LIN {X 0,Y 301.791,Z 514.009,A -85,B 0,C 180,E1 15031.288,E2 15031.288} C_VEL
LIN {X 0,Y 301.177,Z 510.493,A -85,B 0,C 180,E1 15037.195,E2 15037.195} C_VEL
LIN {X 0,Y 300.944,Z 500.832,A -85,B 0,C 180,E1 15043.548,E2 15043.548} C_VEL
LIN {X 0,Y 302.786,Z 486.239,A -85,B 0,C 180,E1 15049.383,E2 15049.383} C_VEL
LIN {X 0,Y 307.108,Z 465.65,A -85,B 0,C 180,E1 15054.908,E2 15054.908} C_VEL
LIN {X 0,Y 312.998,Z 440.583,A -85,B 0,C 180,E1 15059.52,E2 15059.52} C_VEL
LIN {X 0,Y 319.157,Z 413.117,A -85,B 0,C 180,E1 15062.937,E2 15062.937} C_VEL
LIN {X 0,Y 324.854,Z 381.907,A -85,B 0,C 180,E1 15065.445,E2 15065.445} C_VEL
LIN {X 0,Y 326.72,Z 362.395,A -85,B 0,C 180,E1 15066.545,E2 15066.545} C_VEL
LIN {X 0,Y 316.647,Z 334.378,A -85,B 0,C 180,E1 15069.125,E2 15069.125} C_VEL
LIN {X 0,Y 302.51,Z 308.079,A -85,B 0,C 180,E1 15072.331,E2 15072.331} C_VEL
LIN {X 0,Y 294.858,Z 301.001,A -85,B 0,C 180,E1 15074.423,E2 15074.423} C_VEL
LIN {X 0,Y 289.746,Z 297.975,A -85,B 0,C 180,E1 15077.118,E2 15077.118} C_VEL
LIN {X 0,Y 289.332,Z 297.81,A -85,B 0,C 180,E1 15077.961,E2 15077.961} C_VEL
LIN {X 0,Y 289.637,Z 297.81,A -85,B 0,C 180,E1 15086.468,E2 15086.468} C_VEL
LIN {X 0,Y 289.839,Z 297.81,A -85,B 0,C 180,E1 15092.259,E2 15092.259} C_VEL
LIN {X 0,Y 290.263,Z 297.81,A -85,B 0,C 180,E1 15099.35,E2 15099.35} C_VEL
LIN {X 0,Y 290.729,Z 297.81,A -85,B 0,C 180,E1 15108.036,E2 15108.036} C_VEL
LIN {X 0,Y 291.615,Z 297.81,A -85,B 0,C 180,E1 15117.052,E2 15117.052} C_VEL
LIN {X 0,Y 291.518,Z 297.81,A -85,B 0,C 180,E1 15122.986,E2 15122.986} C_VEL
LIN {X 0,Y 290.857,Z 297.81,A -85,B 0,C 180,E1 15131.997,E2 15131.997} C_VEL
LIN {X 0,Y 290.685,Z 297.81,A -85,B 0,C 180,E1 15134.967,E2 15134.967} C_VEL
LIN {X 0,Y 293.021,Z 303.499,A -85,B 0,C 180,E1 15135.796,E2 15135.796} C_VEL
LIN {X 0,Y 305.082,Z 328.065,A -85,B 0,C 180,E1 15139.617,E2 15139.617} C_VEL
LIN {X 0,Y 311.989,Z 352.876,A -85,B 0,C 180,E1 15143.226,E2 15143.226} C_VEL
LIN {X 0,Y 313.291,Z 368.052,A -85,B 0,C 180,E1 15145.499,E2 15145.499} C_VEL
LIN {X 0,Y 307.869,Z 391.312,A -85,B 0,C 180,E1 15149.111,E2 15149.111} C_VEL
LIN {X 0,Y 302.987,Z 408.721,A -85,B 0,C 180,E1 15153.242,E2 15153.242} C_VEL
LIN {X 0,Y 298.665,Z 422.191,A -85,B 0,C 180,E1 15158.382,E2 15158.382} C_VEL
LIN {X 0,Y 296.439,Z 428.527,A -85,B 0,C 180,E1 15162.658,E2 15162.658} C_VEL
LIN {X 0,Y 294.718,Z 431.283,A -85,B 0,C 180,E1 15168.271,E2 15168.271} C_VEL
LIN {X 0,Y 294.669,Z 428.472,A -85,B 0,C 180,E1 15173.6,E2 15173.6} C_VEL
LIN {X 0,Y 296.07,Z 420.423,A -85,B 0,C 180,E1 15178.758,E2 15178.758} C_VEL
LIN {X 0,Y 298.582,Z 406.454,A -85,B 0,C 180,E1 15183.785,E2 15183.785} C_VEL
LIN {X 0,Y 302.074,Z 387.104,A -85,B 0,C 180,E1 15188.21,E2 15188.21} C_VEL
LIN {X 0,Y 305.829,Z 362.988,A -85,B 0,C 180,E1 15191.816,E2 15191.816} C_VEL
LIN {X 0,Y 306.003,Z 353.399,A -85,B 0,C 180,E1 15192.975,E2 15192.975} C_VEL
LIN {X 0,Y 303.879,Z 347.718,A -85,B 0,C 180,E1 15193.781,E2 15193.781} C_VEL
LIN {X 0,Y 302.697,Z 371.6,A -85,B 0,C 180,E1 15196.166,E2 15196.166} C_VEL
LIN {X 0,Y 300.079,Z 393.048,A -85,B 0,C 180,E1 15199.498,E2 15199.498} C_VEL
LIN {X 0,Y 297.619,Z 409.556,A -85,B 0,C 180,E1 15203.45,E2 15203.45} C_VEL
LIN {X 0,Y 295.778,Z 421.095,A -85,B 0,C 180,E1 15207.808,E2 15207.808} C_VEL
LIN {X 0,Y 294.658,Z 428.496,A -85,B 0,C 180,E1 15212.936,E2 15212.936} C_VEL
LIN {X 0,Y 294.506,Z 430.214,A -85,B 0,C 180,E1 15215.883,E2 15215.883} C_VEL
LIN {X 0,Y 294.768,Z 430.176,A -85,B 0,C 180,E1 15218.835,E2 15218.835} C_VEL
LIN {X 0,Y 296.42,Z 425.865,A -85,B 0,C 180,E1 15223.994,E2 15223.994} C_VEL
LIN {X 0,Y 299.258,Z 415.447,A -85,B 0,C 180,E1 15229.134,E2 15229.134} C_VEL
LIN {X 0,Y 302.774,Z 400.098,A -85,B 0,C 180,E1 15233.499,E2 15233.499} C_VEL
LIN {X 0,Y 306.689,Z 379.427,A -85,B 0,C 180,E1 15237.174,E2 15237.174} C_VEL
LIN {X 0,Y 309.289,Z 356.641,A -85,B 0,C 180,E1 15239.755,E2 15239.755} C_VEL
LIN {X 0,Y 303.855,Z 332.82,A -85,B 0,C 180,E1 15242.082,E2 15242.082} C_VEL
LIN {X 0,Y 289.715,Z 297.81,A -85,B 0,C 180,E1 15244.957,E2 15244.957} C_VEL
LIN {X 0,Y 289.4,Z 297.81,A -85,B 0,C 180,E1 15253.085,E2 15253.085} C_VEL
LIN {X 0,Y 289.499,Z 297.81,A -85,B 0,C 180,E1 15261.433,E2 15261.433} C_VEL
LIN {X 0,Y 289.619,Z 297.81,A -85,B 0,C 180,E1 15268.576,E2 15268.576} C_VEL
LIN {X 0,Y 290.019,Z 297.81,A -85,B 0,C 180,E1 15275.381,E2 15275.381} C_VEL
LIN {X 0,Y 290.399,Z 297.81,A -85,B 0,C 180,E1 15281.814,E2 15281.814} C_VEL
LIN {X 0,Y 290.916,Z 297.81,A -85,B 0,C 180,E1 15290.249,E2 15290.249} C_VEL
LIN {X 0,Y 291.631,Z 297.81,A -85,B 0,C 180,E1 15297.015,E2 15297.015} C_VEL
LIN {X 0,Y 291.57,Z 297.81,A -85,B 0,C 180,E1 15302.948,E2 15302.948} C_VEL
LIN {X 0,Y 290.904,Z 297.81,A -85,B 0,C 180,E1 15311.957,E2 15311.957} C_VEL
LIN {X 0,Y 290.36,Z 297.81,A -85,B 0,C 180,E1 15320.695,E2 15320.695} C_VEL
LIN {X 0,Y 289.868,Z 297.81,A -85,B 0,C 180,E1 15327.918,E2 15327.918} C_VEL
LIN {X 0,Y 289.6,Z 297.81,A -85,B 0,C 180,E1 15334.95,E2 15334.95} C_VEL
LIN {X 0,Y 289.442,Z 297.81,A -85,B 0,C 180,E1 15343.122,E2 15343.122} C_VEL
LIN {X 0,Y 289.776,Z 298.498,A -85,B 0,C 180,E1 15350.428,E2 15350.428} C_VEL
LIN {X 0,Y 309.953,Z 350.629,A -85,B 0,C 180,E1 15353.903,E2 15353.903} C_VEL
LIN {X 0,Y 313.87,Z 365.849,A -85,B 0,C 180,E1 15354.929,E2 15354.929} C_VEL
LIN {X 0,Y 309.878,Z 397.751,A -85,B 0,C 180,E1 15356.906,E2 15356.906} C_VEL
LIN {X 0,Y 304.908,Z 427.348,A -85,B 0,C 180,E1 15359.928,E2 15359.928} C_VEL
LIN {X 0,Y 300.107,Z 452.766,A -85,B 0,C 180,E1 15363.792,E2 15363.792} C_VEL
LIN {X 0,Y 295.894,Z 475.187,A -85,B 0,C 180,E1 15368.692,E2 15368.692} C_VEL
LIN {X 0,Y 293.627,Z 492.914,A -85,B 0,C 180,E1 15374.346,E2 15374.346} C_VEL
LIN {X 0,Y 293.234,Z 505.119,A -85,B 0,C 180,E1 15380.371,E2 15380.371} C_VEL
LIN {X 0,Y 293.771,Z 511.106,A -85,B 0,C 180,E1 15385.58,E2 15385.58} C_VEL
LIN {X 0,Y 294.167,Z 512.941,A -85,B 0,C 180,E1 15389.999,E2 15389.999} C_VEL
LIN {X 0,Y 293.543,Z 510.787,A -85,B 0,C 180,E1 15395.9,E2 15395.9} C_VEL
LIN {X 0,Y 292.981,Z 503.359,A -85,B 0,C 180,E1 15401.957,E2 15401.957} C_VEL
LIN {X 0,Y 294.232,Z 490.805,A -85,B 0,C 180,E1 15407.921,E2 15407.921} C_VEL
LIN {X 0,Y 298.019,Z 471.697,A -85,B 0,C 180,E1 15413.895,E2 15413.895} C_VEL
LIN {X 0,Y 304.002,Z 447.808,A -85,B 0,C 180,E1 15418.944,E2 15418.944} C_VEL
LIN {X 0,Y 310.758,Z 420.082,A -85,B 0,C 180,E1 15422.904,E2 15422.904} C_VEL
LIN {X 0,Y 316.915,Z 390.149,A -85,B 0,C 180,E1 15425.689,E2 15425.689} C_VEL
LIN {X 0,Y 320.12,Z 364.362,A -85,B 0,C 180,E1 15427.286,E2 15427.286} C_VEL
LIN {X 0,Y 310.556,Z 337.099,A -85,B 0,C 180,E1 15429.99,E2 15429.99} C_VEL
LIN {X 0,Y 295.545,Z 309.18,A -85,B 0,C 180,E1 15433.663,E2 15433.663} C_VEL
LIN {X 0,Y 289.738,Z 299.386,A -85,B 0,C 180,E1 15435.268,E2 15435.268} C_VEL
LIN {X 0,Y 289.539,Z 297.81,A -85,B 0,C 180,E1 15435.571,E2 15435.571} C_VEL
LIN {X 0,Y 289.332,Z 297.81,A -85,B 0,C 180,E1 15437.961,E2 15437.961} C_VEL
LIN {X 0,Y 286.749,Z 297.81,A -85,B 0,C 180,E1 15440.505,E2 15440.505} C_VEL
LIN {X 0,Y 281.458,Z 297.81,A -85,B 0,C 180,E1 15444.808,E2 15444.808} C_VEL
LIN {X 0,Y 281.799,Z 297.81,A -85,B 0,C 180,E1 15451.209,E2 15451.209} C_VEL
LIN {X 0,Y 282.166,Z 297.81,A -85,B 0,C 180,E1 15458.036,E2 15458.036} C_VEL
LIN {X 0,Y 282.566,Z 297.81,A -85,B 0,C 180,E1 15464.532,E2 15464.532} C_VEL
LIN {X 0,Y 283.042,Z 297.81,A -85,B 0,C 180,E1 15470.816,E2 15470.816} C_VEL
LIN {X 0,Y 283.684,Z 297.81,A -85,B 0,C 180,E1 15476.97,E2 15476.97} C_VEL
LIN {X 0,Y 283.594,Z 297.81,A -85,B 0,C 180,E1 15483.069,E2 15483.069} C_VEL
LIN {X 0,Y 283.112,Z 297.81,A -85,B 0,C 180,E1 15489.221,E2 15489.221} C_VEL
LIN {X 0,Y 282.852,Z 297.81,A -85,B 0,C 180,E1 15493.125,E2 15493.125} C_VEL
LIN {X 0,Y 285.066,Z 303.301,A -85,B 0,C 180,E1 15493.996,E2 15493.996} C_VEL
LIN {X 0,Y 296.674,Z 325.625,A -85,B 0,C 180,E1 15497.88,E2 15497.88} C_VEL
LIN {X 0,Y 304.058,Z 348.441,A -85,B 0,C 180,E1 15501.442,E2 15501.442} C_VEL
LIN {X 0,Y 306.68,Z 369.409,A -85,B 0,C 180,E1 15504.744,E2 15504.744} C_VEL
LIN {X 0,Y 300.833,Z 392.925,A -85,B 0,C 180,E1 15508.507,E2 15508.507} C_VEL
LIN {X 0,Y 295.699,Z 410.151,A -85,B 0,C 180,E1 15512.734,E2 15512.734} C_VEL
LIN {X 0,Y 291.189,Z 423.319,A -85,B 0,C 180,E1 15517.915,E2 15517.915} C_VEL
LIN {X 0,Y 288.516,Z 430.204,A -85,B 0,C 180,E1 15522.928,E2 15522.928} C_VEL
LIN {X 0,Y 287.048,Z 432.419,A -85,B 0,C 180,E1 15527.419,E2 15527.419} C_VEL
LIN {X 0,Y 286.705,Z 430.823,A -85,B 0,C 180,E1 15532.171,E2 15532.171} C_VEL
LIN {X 0,Y 287.863,Z 423.717,A -85,B 0,C 180,E1 15537.767,E2 15537.767} C_VEL
LIN {X 0,Y 290.131,Z 411.587,A -85,B 0,C 180,E1 15542.813,E2 15542.813} C_VEL
LIN {X 0,Y 293.356,Z 394.666,A -85,B 0,C 180,E1 15547.289,E2 15547.289} C_VEL
LIN {X 0,Y 297.189,Z 372.469,A -85,B 0,C 180,E1 15551.203,E2 15551.203} C_VEL
LIN {X 0,Y 298.833,Z 356.279,A -85,B 0,C 180,E1 15553.285,E2 15553.285} C_VEL
LIN {X 0,Y 296.944,Z 353.965,A -85,B 0,C 180,E1 15553.766,E2 15553.766} C_VEL
LIN {X 0,Y 294.567,Z 378.458,A -85,B 0,C 180,E1 15556.486,E2 15556.486} C_VEL
LIN {X 0,Y 291.698,Z 399.409,A -85,B 0,C 180,E1 15560.241,E2 15560.241} C_VEL
LIN {X 0,Y 289.176,Z 415.34,A -85,B 0,C 180,E1 15564.761,E2 15564.761} C_VEL
LIN {X 0,Y 287.366,Z 426.199,A -85,B 0,C 180,E1 15570.001,E2 15570.001} C_VEL
LIN {X 0,Y 286.828,Z 429.651,A -85,B 0,C 180,E1 15573.017,E2 15573.017} C_VEL
LIN {X 0,Y 286.689,Z 431.329,A -85,B 0,C 180,E1 15576.044,E2 15576.044} C_VEL
LIN {X 0,Y 287.015,Z 431.225,A -85,B 0,C 180,E1 15579.076,E2 15579.076} C_VEL
LIN {X 0,Y 288.731,Z 426.889,A -85,B 0,C 180,E1 15584.318,E2 15584.318} C_VEL
LIN {X 0,Y 291.271,Z 418.194,A -85,B 0,C 180,E1 15588.893,E2 15588.893} C_VEL
LIN {X 0,Y 295.038,Z 402.907,A -85,B 0,C 180,E1 15593.602,E2 15593.602} C_VEL
LIN {X 0,Y 299.062,Z 383.23,A -85,B 0,C 180,E1 15597.366,E2 15597.366} C_VEL
LIN {X 0,Y 302.392,Z 360.317,A -85,B 0,C 180,E1 15600.134,E2 15600.134} C_VEL
LIN {X 0,Y 297.677,Z 337.372,A -85,B 0,C 180,E1 15602.53,E2 15602.53} C_VEL
LIN {X 0,Y 285.512,Z 307.036,A -85,B 0,C 180,E1 15605.099,E2 15605.099} C_VEL
LIN {X 0,Y 281.647,Z 297.81,A -85,B 0,C 180,E1 15605.978,E2 15605.978} C_VEL
LIN {X 0,Y 281.379,Z 297.81,A -85,B 0,C 180,E1 15614.202,E2 15614.202} C_VEL
LIN {X 0,Y 281.401,Z 297.81,A -85,B 0,C 180,E1 15619.921,E2 15619.921} C_VEL
LIN {X 0,Y 281.677,Z 297.81,A -85,B 0,C 180,E1 15627.583,E2 15627.583} C_VEL
LIN {X 0,Y 282.132,Z 297.81,A -85,B 0,C 180,E1 15635.404,E2 15635.404} C_VEL
LIN {X 0,Y 282.555,Z 297.81,A -85,B 0,C 180,E1 15644.01,E2 15644.01} C_VEL
LIN {X 0,Y 283.082,Z 297.81,A -85,B 0,C 180,E1 15650.778,E2 15650.778} C_VEL
LIN {X 0,Y 283.701,Z 297.81,A -85,B 0,C 180,E1 15656.932,E2 15656.932} C_VEL
LIN {X 0,Y 283.645,Z 297.81,A -85,B 0,C 180,E1 15663.031,E2 15663.031} C_VEL
LIN {X 0,Y 283.152,Z 297.81,A -85,B 0,C 180,E1 15669.181,E2 15669.181} C_VEL
LIN {X 0,Y 282.614,Z 297.81,A -85,B 0,C 180,E1 15676.031,E2 15676.031} C_VEL
LIN {X 0,Y 282.143,Z 297.81,A -85,B 0,C 180,E1 15684.601,E2 15684.601} C_VEL
LIN {X 0,Y 281.742,Z 297.81,A -85,B 0,C 180,E1 15692.363,E2 15692.363} C_VEL
LIN {X 0,Y 281.432,Z 297.81,A -85,B 0,C 180,E1 15701.351,E2 15701.351} C_VEL
LIN {X 0,Y 281.777,Z 297.81,A -85,B 0,C 180,E1 15709.488,E2 15709.488} C_VEL
LIN {X 0,Y 302.846,Z 352.489,A -85,B 0,C 180,E1 15713.315,E2 15713.315} C_VEL
LIN {X 0,Y 306.58,Z 367.201,A -85,B 0,C 180,E1 15714.371,E2 15714.371} C_VEL
LIN {X 0,Y 302.451,Z 398.701,A -85,B 0,C 180,E1 15716.422,E2 15716.422} C_VEL
LIN {X 0,Y 297.175,Z 428.783,A -85,B 0,C 180,E1 15719.648,E2 15719.648} C_VEL
LIN {X 0,Y 291.863,Z 455.219,A -85,B 0,C 180,E1 15723.929,E2 15723.929} C_VEL
LIN {X 0,Y 287.627,Z 477.566,A -85,B 0,C 180,E1 15729.24,E2 15729.24} C_VEL
LIN {X 0,Y 285.642,Z 493.29,A -85,B 0,C 180,E1 15734.683,E2 15734.683} C_VEL
LIN {X 0,Y 285.406,Z 504.98,A -85,B 0,C 180,E1 15740.873,E2 15740.873} C_VEL
LIN {X 0,Y 285.932,Z 509.912,A -85,B 0,C 180,E1 15745.459,E2 15745.459} C_VEL
LIN {X 0,Y 286.352,Z 511.824,A -85,B 0,C 180,E1 15749.999,E2 15749.999} C_VEL
LIN {X 0,Y 286.049,Z 511.441,A -85,B 0,C 180,E1 15753.023,E2 15753.023} C_VEL
LIN {X 0,Y 285.263,Z 506.719,A -85,B 0,C 180,E1 15759.13,E2 15759.13} C_VEL
LIN {X 0,Y 285.53,Z 496.88,A -85,B 0,C 180,E1 15765.321,E2 15765.321} C_VEL
LIN {X 0,Y 288.492,Z 480.067,A -85,B 0,C 180,E1 15771.88,E2 15771.88} C_VEL
LIN {X 0,Y 293.941,Z 458.261,A -85,B 0,C 180,E1 15777.517,E2 15777.517} C_VEL
LIN {X 0,Y 300.68,Z 432.847,A -85,B 0,C 180,E1 15781.984,E2 15781.984} C_VEL
LIN {X 0,Y 307.715,Z 403.515,A -85,B 0,C 180,E1 15785.398,E2 15785.398} C_VEL
LIN {X 0,Y 313.552,Z 371.306,A -85,B 0,C 180,E1 15787.722,E2 15787.722} C_VEL
LIN {X 0,Y 313.18,Z 364.985,A -85,B 0,C 180,E1 15788.214,E2 15788.214} C_VEL
LIN {X 0,Y 304.443,Z 339.762,A -85,B 0,C 180,E1 15790.922,E2 15790.922} C_VEL
LIN {X 0,Y 290.715,Z 314.15,A -85,B 0,C 180,E1 15794.487,E2 15794.487} C_VEL
LIN {X 0,Y 283.669,Z 303.218,A -85,B 0,C 180,E1 15796.549,E2 15796.549} C_VEL
LIN {X 0,Y 281.52,Z 297.81,A -85,B 0,C 180,E1 15797.338,E2 15797.338} C_VEL
LIN {X 0,Y 281.458,Z 297.81,A -85,B 0,C 180,E1 15804.808,E2 15804.808} C_VEL
LIN {X 0,Y 279.049,Z 297.81,A -85,B 0,C 180,E1 15807.427,E2 15807.427} C_VEL
LIN {X 0,Y 273.871,Z 297.81,A -85,B 0,C 180,E1 15811.859,E2 15811.859} C_VEL
LIN {X 0,Y 274.257,Z 297.81,A -85,B 0,C 180,E1 15819.284,E2 15819.284} C_VEL
LIN {X 0,Y 274.794,Z 297.81,A -85,B 0,C 180,E1 15827.331,E2 15827.331} C_VEL
LIN {X 0,Y 275.365,Z 297.81,A -85,B 0,C 180,E1 15833.727,E2 15833.727} C_VEL
LIN {X 0,Y 275.921,Z 297.81,A -85,B 0,C 180,E1 15840.02,E2 15840.02} C_VEL
LIN {X 0,Y 275.224,Z 297.81,A -85,B 0,C 180,E1 15849.29,E2 15849.29} C_VEL
LIN {X 0,Y 275.008,Z 298.149,A -85,B 0,C 180,E1 15851.091,E2 15851.091} C_VEL
LIN {X 0,Y 277.4,Z 303.463,A -85,B 0,C 180,E1 15852.06,E2 15852.06} C_VEL
LIN {X 0,Y 288.452,Z 323.451,A -85,B 0,C 180,E1 15856.024,E2 15856.024} C_VEL
LIN {X 0,Y 296.621,Z 346.543,A -85,B 0,C 180,E1 15859.91,E2 15859.91} C_VEL
LIN {X 0,Y 300.124,Z 369.507,A -85,B 0,C 180,E1 15863.738,E2 15863.738} C_VEL
LIN {X 0,Y 294.43,Z 392.663,A -85,B 0,C 180,E1 15867.49,E2 15867.49} C_VEL
LIN {X 0,Y 289.022,Z 409.878,A -85,B 0,C 180,E1 15871.675,E2 15871.675} C_VEL
LIN {X 0,Y 284.51,Z 422.433,A -85,B 0,C 180,E1 15876.38,E2 15876.38} C_VEL
LIN {X 0,Y 281.403,Z 430.156,A -85,B 0,C 180,E1 15881.347,E2 15881.347} C_VEL
LIN {X 0,Y 279.75,Z 433.129,A -85,B 0,C 180,E1 15885.475,E2 15885.475} C_VEL
LIN {X 0,Y 278.854,Z 432.696,A -85,B 0,C 180,E1 15890.907,E2 15890.907} C_VEL
LIN {X 0,Y 279.687,Z 426.762,A -85,B 0,C 180,E1 15896.704,E2 15896.704} C_VEL
LIN {X 0,Y 281.935,Z 415.187,A -85,B 0,C 180,E1 15902.173,E2 15902.173} C_VEL
LIN {X 0,Y 285.175,Z 398.75,A -85,B 0,C 180,E1 15906.979,E2 15906.979} C_VEL
LIN {X 0,Y 289.128,Z 377.292,A -85,B 0,C 180,E1 15911.11,E2 15911.11} C_VEL
LIN {X 0,Y 291.378,Z 363.262,A -85,B 0,C 180,E1 15913.065,E2 15913.065} C_VEL
LIN {X 0,Y 289.197,Z 360.16,A -85,B 0,C 180,E1 15913.713,E2 15913.713} C_VEL
LIN {X 0,Y 286.517,Z 383.805,A -85,B 0,C 180,E1 15916.679,E2 15916.679} C_VEL
LIN {X 0,Y 283.656,Z 403.2,A -85,B 0,C 180,E1 15920.533,E2 15920.533} C_VEL
LIN {X 0,Y 281.397,Z 416.682,A -85,B 0,C 180,E1 15924.616,E2 15924.616} C_VEL
LIN {X 0,Y 279.532,Z 427.42,A -85,B 0,C 180,E1 15930.001,E2 15930.001} C_VEL
LIN {X 0,Y 278.989,Z 430.807,A -85,B 0,C 180,E1 15933.101,E2 15933.101} C_VEL
LIN {X 0,Y 278.866,Z 432.437,A -85,B 0,C 180,E1 15936.214,E2 15936.214} C_VEL
LIN {X 0,Y 279.242,Z 432.277,A -85,B 0,C 180,E1 15939.331,E2 15939.331} C_VEL
LIN {X 0,Y 281.209,Z 427.535,A -85,B 0,C 180,E1 15944.925,E2 15944.925} C_VEL
LIN {X 0,Y 284.336,Z 417.08,A -85,B 0,C 180,E1 15950.18,E2 15950.18} C_VEL
LIN {X 0,Y 288.308,Z 401.414,A -85,B 0,C 180,E1 15954.755,E2 15954.755} C_VEL
LIN {X 0,Y 292.539,Z 380.963,A -85,B 0,C 180,E1 15958.491,E2 15958.491} C_VEL
LIN {X 0,Y 295.194,Z 360.337,A -85,B 0,C 180,E1 15960.949,E2 15960.949} C_VEL
LIN {X 0,Y 289.798,Z 336.185,A -85,B 0,C 180,E1 15963.542,E2 15963.542} C_VEL
LIN {X 0,Y 277.11,Z 306.368,A -85,B 0,C 180,E1 15966.232,E2 15966.232} C_VEL
LIN {X 0,Y 273.604,Z 297.81,A -85,B 0,C 180,E1 15967.086,E2 15967.086} C_VEL
LIN {X 0,Y 273.468,Z 297.81,A -85,B 0,C 180,E1 15975.836,E2 15975.836} C_VEL
LIN {X 0,Y 273.461,Z 297.81,A -85,B 0,C 180,E1 15982.601,E2 15982.601} C_VEL
LIN {X 0,Y 273.808,Z 297.81,A -85,B 0,C 180,E1 15990.24,E2 15990.24} C_VEL
LIN {X 0,Y 274.292,Z 297.81,A -85,B 0,C 180,E1 15999.27,E2 15999.27} C_VEL
LIN {X 0,Y 274.844,Z 297.81,A -85,B 0,C 180,E1 16007.293,E2 16007.293} C_VEL
LIN {X 0,Y 275.393,Z 297.81,A -85,B 0,C 180,E1 16013.688,E2 16013.688} C_VEL
LIN {X 0,Y 276.036,Z 297.81,A -85,B 0,C 180,E1 16019.98,E2 16019.98} C_VEL
LIN {X 0,Y 275.2,Z 297.81,A -85,B 0,C 180,E1 16029.449,E2 16029.449} C_VEL
LIN {X 0,Y 274.728,Z 297.81,A -85,B 0,C 180,E1 16035.92,E2 16035.92} C_VEL
LIN {X 0,Y 274.265,Z 297.81,A -85,B 0,C 180,E1 16042.632,E2 16042.632} C_VEL
LIN {X 0,Y 273.874,Z 297.81,A -85,B 0,C 180,E1 16049.706,E2 16049.706} C_VEL
LIN {X 0,Y 273.506,Z 297.81,A -85,B 0,C 180,E1 16057.342,E2 16057.342} C_VEL
LIN {X 0,Y 273.573,Z 297.81,A -85,B 0,C 180,E1 16065.786,E2 16065.786} C_VEL
LIN {X 0,Y 273.819,Z 297.81,A -85,B 0,C 180,E1 16068.497,E2 16068.497} C_VEL
LIN {X 0,Y 295.092,Z 352.338,A -85,B 0,C 180,E1 16072.563,E2 16072.563} C_VEL
LIN {X 0,Y 299.245,Z 369.351,A -85,B 0,C 180,E1 16073.843,E2 16073.843} C_VEL
LIN {X 0,Y 294.934,Z 400.043,A -85,B 0,C 180,E1 16075.971,E2 16075.971} C_VEL
LIN {X 0,Y 289.575,Z 429.128,A -85,B 0,C 180,E1 16079.223,E2 16079.223} C_VEL
LIN {X 0,Y 284.164,Z 455.141,A -85,B 0,C 180,E1 16083.593,E2 16083.593} C_VEL
LIN {X 0,Y 279.809,Z 477.301,A -85,B 0,C 180,E1 16089.066,E2 16089.066} C_VEL
LIN {X 0,Y 277.691,Z 493.638,A -85,B 0,C 180,E1 16095.041,E2 16095.041} C_VEL
LIN {X 0,Y 277.595,Z 504.699,A -85,B 0,C 180,E1 16101.402,E2 16101.402} C_VEL
LIN {X 0,Y 278.299,Z 509.701,A -85,B 0,C 180,E1 16106.891,E2 16106.891} C_VEL
LIN {X 0,Y 278.524,Z 510.7,A -85,B 0,C 180,E1 16109.999,E2 16109.999} C_VEL
LIN {X 0,Y 278.197,Z 510.343,A -85,B 0,C 180,E1 16113.108,E2 16113.108} C_VEL
LIN {X 0,Y 277.346,Z 505.67,A -85,B 0,C 180,E1 16119.393,E2 16119.393} C_VEL
LIN {X 0,Y 277.724,Z 495.895,A -85,B 0,C 180,E1 16125.763,E2 16125.763} C_VEL
LIN {X 0,Y 280.964,Z 479.199,A -85,B 0,C 180,E1 16132.485,E2 16132.485} C_VEL
LIN {X 0,Y 286.783,Z 457.502,A -85,B 0,C 180,E1 16138.265,E2 16138.265} C_VEL
LIN {X 0,Y 293.959,Z 432.034,A -85,B 0,C 180,E1 16142.833,E2 16142.833} C_VEL
LIN {X 0,Y 301.26,Z 403.104,A -85,B 0,C 180,E1 16146.275,E2 16146.275} C_VEL
LIN {X 0,Y 307.338,Z 371.242,A -85,B 0,C 180,E1 16148.624,E2 16148.624} C_VEL
LIN {X 0,Y 301.194,Z 349.042,A -85,B 0,C 180,E1 16151.067,E2 16151.067} C_VEL
LIN {X 0,Y 288.211,Z 322.64,A -85,B 0,C 180,E1 16154.706,E2 16154.706} C_VEL
LIN {X 0,Y 276.575,Z 304.046,A -85,B 0,C 180,E1 16158.362,E2 16158.362} C_VEL
LIN {X 0,Y 273.66,Z 299.357,A -85,B 0,C 180,E1 16159.406,E2 16159.406} C_VEL
LIN {X 0,Y 273.505,Z 297.81,A -85,B 0,C 180,E1 16159.647,E2 16159.647} C_VEL
LIN {X 0,Y 273.635,Z 297.81,A -85,B 0,C 180,E1 16166.555,E2 16166.555} C_VEL
LIN {X 0,Y 273.871,Z 297.81,A -85,B 0,C 180,E1 16171.859,E2 16171.859} C_VEL
LIN {X 0,Y 271.322,Z 297.81,A -85,B 0,C 180,E1 16174.572,E2 16174.572} C_VEL
LIN {X 0,Y 266.238,Z 297.81,A -85,B 0,C 180,E1 16179.168,E2 16179.168} C_VEL
LIN {X 0,Y 266.821,Z 297.81,A -85,B 0,C 180,E1 16186.946,E2 16186.946} C_VEL
LIN {X 0,Y 267.424,Z 297.81,A -85,B 0,C 180,E1 16193.54,E2 16193.54} C_VEL
LIN {X 0,Y 268.014,Z 297.81,A -85,B 0,C 180,E1 16200.02,E2 16200.02} C_VEL
LIN {X 0,Y 267.307,Z 297.81,A -85,B 0,C 180,E1 16208.683,E2 16208.683} C_VEL
LIN {X 0,Y 269.585,Z 303.422,A -85,B 0,C 180,E1 16209.789,E2 16209.789} C_VEL
LIN {X 0,Y 278.977,Z 319.201,A -85,B 0,C 180,E1 16213.472,E2 16213.472} C_VEL
LIN {X 0,Y 288.438,Z 342.011,A -85,B 0,C 180,E1 16217.789,E2 16217.789} C_VEL
LIN {X 0,Y 292.923,Z 364.093,A -85,B 0,C 180,E1 16221.632,E2 16221.632} C_VEL
LIN {X 0,Y 292.974,Z 375.24,A -85,B 0,C 180,E1 16223.547,E2 16223.547} C_VEL
LIN {X 0,Y 286.411,Z 397.791,A -85,B 0,C 180,E1 16227.545,E2 16227.545} C_VEL
LIN {X 0,Y 280.635,Z 414.67,A -85,B 0,C 180,E1 16232.171,E2 16232.171} C_VEL
LIN {X 0,Y 275.808,Z 426.847,A -85,B 0,C 180,E1 16237.603,E2 16237.603} C_VEL
LIN {X 0,Y 273.52,Z 431.879,A -85,B 0,C 180,E1 16241.483,E2 16241.483} C_VEL
LIN {X 0,Y 271.696,Z 434.557,A -85,B 0,C 180,E1 16246.252,E2 16246.252} C_VEL
LIN {X 0,Y 271.151,Z 432.168,A -85,B 0,C 180,E1 16253.146,E2 16253.146} C_VEL
LIN {X 0,Y 272.729,Z 423.507,A -85,B 0,C 180,E1 16259.28,E2 16259.28} C_VEL
LIN {X 0,Y 275.404,Z 410.394,A -85,B 0,C 180,E1 16264.442,E2 16264.442} C_VEL
LIN {X 0,Y 279.298,Z 391.265,A -85,B 0,C 180,E1 16269.259,E2 16269.259} C_VEL
LIN {X 0,Y 283.411,Z 368.522,A -85,B 0,C 180,E1 16273.058,E2 16273.058} C_VEL
LIN {X 0,Y 281.302,Z 366.516,A -85,B 0,C 180,E1 16273.728,E2 16273.728} C_VEL
LIN {X 0,Y 278.314,Z 389.906,A -85,B 0,C 180,E1 16277.077,E2 16277.077} C_VEL
LIN {X 0,Y 275.332,Z 408.596,A -85,B 0,C 180,E1 16281.332,E2 16281.332} C_VEL
LIN {X 0,Y 272.913,Z 421.74,A -85,B 0,C 180,E1 16286.038,E2 16286.038} C_VEL
LIN {X 0,Y 271.396,Z 430.54,A -85,B 0,C 180,E1 16291.594,E2 16291.594} C_VEL
LIN {X 0,Y 271.049,Z 433.537,A -85,B 0,C 180,E1 16296.394,E2 16296.394} C_VEL
LIN {X 0,Y 271.491,Z 433.327,A -85,B 0,C 180,E1 16299.6,E2 16299.6} C_VEL
LIN {X 0,Y 273.362,Z 429.156,A -85,B 0,C 180,E1 16304.852,E2 16304.852} C_VEL
LIN {X 0,Y 276.33,Z 419.884,A -85,B 0,C 180,E1 16309.957,E2 16309.957} C_VEL
LIN {X 0,Y 280.444,Z 404.981,A -85,B 0,C 180,E1 16314.718,E2 16314.718} C_VEL
LIN {X 0,Y 284.633,Z 386.282,A -85,B 0,C 180,E1 16318.5,E2 16318.5} C_VEL
LIN {X 0,Y 288.298,Z 363.539,A -85,B 0,C 180,E1 16321.425,E2 16321.425} C_VEL
LIN {X 0,Y 283.612,Z 340.371,A -85,B 0,C 180,E1 16324.067,E2 16324.067} C_VEL
LIN {X 0,Y 272.3,Z 312.387,A -85,B 0,C 180,E1 16326.721,E2 16326.721} C_VEL
LIN {X 0,Y 265.592,Z 297.81,A -85,B 0,C 180,E1 16328.305,E2 16328.305} C_VEL
LIN {X 0,Y 265.529,Z 297.81,A -85,B 0,C 180,E1 16336.974,E2 16336.974} C_VEL
LIN {X 0,Y 265.597,Z 297.81,A -85,B 0,C 180,E1 16345.353,E2 16345.353} C_VEL
LIN {X 0,Y 265.986,Z 297.81,A -85,B 0,C 180,E1 16352.985,E2 16352.985} C_VEL
LIN {X 0,Y 266.451,Z 297.81,A -85,B 0,C 180,E1 16360.113,E2 16360.113} C_VEL
LIN {X 0,Y 266.873,Z 297.81,A -85,B 0,C 180,E1 16366.907,E2 16366.907} C_VEL
LIN {X 0,Y 267.453,Z 297.81,A -85,B 0,C 180,E1 16373.5,E2 16373.5} C_VEL
LIN {X 0,Y 268.128,Z 297.81,A -85,B 0,C 180,E1 16379.98,E2 16379.98} C_VEL
LIN {X 0,Y 267.481,Z 297.81,A -85,B 0,C 180,E1 16386.458,E2 16386.458} C_VEL
LIN {X 0,Y 266.991,Z 297.81,A -85,B 0,C 180,E1 16393.046,E2 16393.046} C_VEL
LIN {X 0,Y 266.492,Z 297.81,A -85,B 0,C 180,E1 16399.841,E2 16399.841} C_VEL
LIN {X 0,Y 266.011,Z 297.81,A -85,B 0,C 180,E1 16406.967,E2 16406.967} C_VEL
LIN {X 0,Y 265.66,Z 297.81,A -85,B 0,C 180,E1 16414.589,E2 16414.589} C_VEL
LIN {X 0,Y 265.587,Z 297.81,A -85,B 0,C 180,E1 16422.959,E2 16422.959} C_VEL
LIN {X 0,Y 265.766,Z 297.916,A -85,B 0,C 180,E1 16427.544,E2 16427.544} C_VEL
LIN {X 0,Y 287.407,Z 352.313,A -85,B 0,C 180,E1 16431.778,E2 16431.778} C_VEL
LIN {X 0,Y 292.004,Z 370.477,A -85,B 0,C 180,E1 16433.24,E2 16433.24} C_VEL
LIN {X 0,Y 287.229,Z 402.531,A -85,B 0,C 180,E1 16435.613,E2 16435.613} C_VEL
LIN {X 0,Y 281.418,Z 431.954,A -85,B 0,C 180,E1 16439.155,E2 16439.155} C_VEL
LIN {X 0,Y 276.038,Z 456.758,A -85,B 0,C 180,E1 16443.629,E2 16443.629} C_VEL
LIN {X 0,Y 271.74,Z 478.163,A -85,B 0,C 180,E1 16449.266,E2 16449.266} C_VEL
LIN {X 0,Y 269.756,Z 493.932,A -85,B 0,C 180,E1 16455.419,E2 16455.419} C_VEL
LIN {X 0,Y 269.828,Z 504.415,A -85,B 0,C 180,E1 16461.962,E2 16461.962} C_VEL
LIN {X 0,Y 270.455,Z 508.519,A -85,B 0,C 180,E1 16466.801,E2 16466.801} C_VEL
LIN {X 0,Y 270.722,Z 509.579,A -85,B 0,C 180,E1 16469.999,E2 16469.999} C_VEL
LIN {X 0,Y 270.332,Z 509.234,A -85,B 0,C 180,E1 16473.199,E2 16473.199} C_VEL
LIN {X 0,Y 269.466,Z 504.635,A -85,B 0,C 180,E1 16479.671,E2 16479.671} C_VEL
LIN {X 0,Y 270.117,Z 493.686,A -85,B 0,C 180,E1 16486.858,E2 16486.858} C_VEL
LIN {X 0,Y 273.711,Z 477.349,A -85,B 0,C 180,E1 16493.464,E2 16493.464} C_VEL
LIN {X 0,Y 279.697,Z 456.738,A -85,B 0,C 180,E1 16499.048,E2 16499.048} C_VEL
LIN {X 0,Y 287.234,Z 431.473,A -85,B 0,C 180,E1 16503.703,E2 16503.703} C_VEL
LIN {X 0,Y 294.896,Z 402.74,A -85,B 0,C 180,E1 16507.188,E2 16507.188} C_VEL
LIN {X 0,Y 300.892,Z 371.688,A -85,B 0,C 180,E1 16509.577,E2 16509.577} C_VEL
LIN {X 0,Y 293.59,Z 347.701,A -85,B 0,C 180,E1 16512.527,E2 16512.527} C_VEL
LIN {X 0,Y 280.155,Z 321.431,A -85,B 0,C 180,E1 16516.651,E2 16516.651} C_VEL
LIN {X 0,Y 268.475,Z 303.948,A -85,B 0,C 180,E1 16520.776,E2 16520.776} C_VEL
LIN {X 0,Y 265.627,Z 298.934,A -85,B 0,C 180,E1 16521.996,E2 16521.996} C_VEL
LIN {X 0,Y 265.574,Z 297.81,A -85,B 0,C 180,E1 16522.446,E2 16522.446} C_VEL
LIN {X 0,Y 265.775,Z 297.81,A -85,B 0,C 180,E1 16529.292,E2 16529.292} C_VEL
LIN {X 0,Y 266.179,Z 297.81,A -85,B 0,C 180,E1 16536.641,E2 16536.641} C_VEL
LIN {X 0,Y 266.238,Z 297.81,A -85,B 0,C 180,E1 16539.168,E2 16539.168} C_VEL
LIN {X 0,Y 264.072,Z 297.81,A -85,B 0,C 180,E1 16541.953,E2 16541.953} C_VEL
LIN {X 0,Y 258.879,Z 297.81,A -85,B 0,C 180,E1 16546.674,E2 16546.674} C_VEL
LIN {X 0,Y 259.474,Z 297.81,A -85,B 0,C 180,E1 16553.341,E2 16553.341} C_VEL
LIN {X 0,Y 260.106,Z 297.81,A -85,B 0,C 180,E1 16560.021,E2 16560.021} C_VEL
LIN {X 0,Y 259.571,Z 297.883,A -85,B 0,C 180,E1 16565.86,E2 16565.86} C_VEL
LIN {X 0,Y 261.491,Z 303.044,A -85,B 0,C 180,E1 16566.992,E2 16566.992} C_VEL
LIN {X 0,Y 264.165,Z 306.401,A -85,B 0,C 180,E1 16568.206,E2 16568.206} C_VEL
LIN {X 0,Y 275.569,Z 326.661,A -85,B 0,C 180,E1 16573.205,E2 16573.205} C_VEL
LIN {X 0,Y 283.292,Z 348.205,A -85,B 0,C 180,E1 16577.454,E2 16577.454} C_VEL
LIN {X 0,Y 286.745,Z 370.855,A -85,B 0,C 180,E1 16581.636,E2 16581.636} C_VEL
LIN {X 0,Y 285.636,Z 379.889,A -85,B 0,C 180,E1 16583.169,E2 16583.169} C_VEL
LIN {X 0,Y 278.979,Z 401.075,A -85,B 0,C 180,E1 16587.211,E2 16587.211} C_VEL
LIN {X 0,Y 272.678,Z 417.898,A -85,B 0,C 180,E1 16592.237,E2 16592.237} C_VEL
LIN {X 0,Y 267.782,Z 429.298,A -85,B 0,C 180,E1 16597.917,E2 16597.917} C_VEL
LIN {X 0,Y 264.948,Z 434.582,A -85,B 0,C 180,E1 16603.144,E2 16603.144} C_VEL
LIN {X 0,Y 263.487,Z 435.76,A -85,B 0,C 180,E1 16608.15,E2 16608.15} C_VEL
LIN {X 0,Y 263.343,Z 433.024,A -85,B 0,C 180,E1 16613.38,E2 16613.38} C_VEL
LIN {X 0,Y 264.827,Z 425.093,A -85,B 0,C 180,E1 16619.149,E2 16619.149} C_VEL
LIN {X 0,Y 267.562,Z 412.143,A -85,B 0,C 180,E1 16624.522,E2 16624.522} C_VEL
LIN {X 0,Y 271.56,Z 393.392,A -85,B 0,C 180,E1 16629.479,E2 16629.479} C_VEL
LIN {X 0,Y 274.804,Z 372.608,A -85,B 0,C 180,E1 16633.246,E2 16633.246} C_VEL
LIN {X 0,Y 273.498,Z 371.778,A -85,B 0,C 180,E1 16633.679,E2 16633.679} C_VEL
LIN {X 0,Y 270.462,Z 393.508,A -85,B 0,C 180,E1 16637.105,E2 16637.105} C_VEL
LIN {X 0,Y 267.323,Z 411.839,A -85,B 0,C 180,E1 16641.643,E2 16641.643} C_VEL
LIN {X 0,Y 264.808,Z 424.675,A -85,B 0,C 180,E1 16646.734,E2 16646.734} C_VEL
LIN {X 0,Y 263.575,Z 431.714,A -85,B 0,C 180,E1 16651.641,E2 16651.641} C_VEL
LIN {X 0,Y 263.232,Z 434.632,A -85,B 0,C 180,E1 16656.584,E2 16656.584} C_VEL
LIN {X 0,Y 264.216,Z 433.6,A -85,B 0,C 180,E1 16661.532,E2 16661.532} C_VEL
LIN {X 0,Y 266.792,Z 427.234,A -85,B 0,C 180,E1 16667.275,E2 16667.275} C_VEL
LIN {X 0,Y 270.504,Z 415.399,A -85,B 0,C 180,E1 16672.553,E2 16672.553} C_VEL
LIN {X 0,Y 274.911,Z 399.231,A -85,B 0,C 180,E1 16676.927,E2 16676.927} C_VEL
LIN {X 0,Y 279.383,Z 378.287,A -85,B 0,C 180,E1 16680.537,E2 16680.537} C_VEL
LIN {X 0,Y 281.038,Z 362.366,A -85,B 0,C 180,E1 16682.476,E2 16682.476} C_VEL
LIN {X 0,Y 275.582,Z 338.585,A -85,B 0,C 180,E1 16685.256,E2 16685.256} C_VEL
LIN {X 0,Y 262.275,Z 308.128,A -85,B 0,C 180,E1 16688.36,E2 16688.36} C_VEL
LIN {X 0,Y 257.58,Z 297.81,A -85,B 0,C 180,E1 16689.671,E2 16689.671} C_VEL
LIN {X 0,Y 257.476,Z 297.81,A -85,B 0,C 180,E1 16695.277,E2 16695.277} C_VEL
LIN {X 0,Y 257.615,Z 297.81,A -85,B 0,C 180,E1 16704.116,E2 16704.116} C_VEL
LIN {X 0,Y 257.917,Z 297.81,A -85,B 0,C 180,E1 16712.067,E2 16712.067} C_VEL
LIN {X 0,Y 258.429,Z 297.81,A -85,B 0,C 180,E1 16719.469,E2 16719.469} C_VEL
LIN {X 0,Y 258.938,Z 297.81,A -85,B 0,C 180,E1 16726.498,E2 16726.498} C_VEL
LIN {X 0,Y 259.502,Z 297.81,A -85,B 0,C 180,E1 16733.432,E2 16733.432} C_VEL
LIN {X 0,Y 260.219,Z 297.81,A -85,B 0,C 180,E1 16739.979,E2 16739.979} C_VEL
LIN {X 0,Y 259.346,Z 297.81,A -85,B 0,C 180,E1 16748.446,E2 16748.446} C_VEL
LIN {X 0,Y 258.742,Z 297.81,A -85,B 0,C 180,E1 16756.933,E2 16756.933} C_VEL
LIN {X 0,Y 258.243,Z 297.81,A -85,B 0,C 180,E1 16764.122,E2 16764.122} C_VEL
LIN {X 0,Y 257.808,Z 297.81,A -85,B 0,C 180,E1 16771.765,E2 16771.765} C_VEL
LIN {X 0,Y 257.537,Z 297.81,A -85,B 0,C 180,E1 16780.383,E2 16780.383} C_VEL
LIN {X 0,Y 257.714,Z 297.81,A -85,B 0,C 180,E1 16786.467,E2 16786.467} C_VEL
LIN {X 0,Y 278.795,Z 349.569,A -85,B 0,C 180,E1 16790.747,E2 16790.747} C_VEL
LIN {X 0,Y 284.759,Z 371.949,A -85,B 0,C 180,E1 16792.631,E2 16792.631} C_VEL
LIN {X 0,Y 279.844,Z 403.041,A -85,B 0,C 180,E1 16795.044,E2 16795.044} C_VEL
LIN {X 0,Y 273.806,Z 432.344,A -85,B 0,C 180,E1 16798.719,E2 16798.719} C_VEL
LIN {X 0,Y 267.956,Z 458.32,A -85,B 0,C 180,E1 16803.664,E2 16803.664} C_VEL
LIN {X 0,Y 263.657,Z 478.957,A -85,B 0,C 180,E1 16809.478,E2 16809.478} C_VEL
LIN {X 0,Y 261.816,Z 494.089,A -85,B 0,C 180,E1 16815.82,E2 16815.82} C_VEL
LIN {X 0,Y 261.955,Z 503.128,A -85,B 0,C 180,E1 16821.719,E2 16821.719} C_VEL
LIN {X 0,Y 262.609,Z 507.333,A -85,B 0,C 180,E1 16826.705,E2 16826.705} C_VEL
LIN {X 0,Y 262.891,Z 508.452,A -85,B 0,C 180,E1 16829.999,E2 16829.999} C_VEL
LIN {X 0,Y 262.474,Z 508.125,A -85,B 0,C 180,E1 16833.295,E2 16833.295} C_VEL
LIN {X 0,Y 261.556,Z 503.605,A -85,B 0,C 180,E1 16839.966,E2 16839.966} C_VEL
LIN {X 0,Y 262.351,Z 492.862,A -85,B 0,C 180,E1 16847.312,E2 16847.312} C_VEL
LIN {X 0,Y 266.121,Z 477.071,A -85,B 0,C 180,E1 16853.969,E2 16853.969} C_VEL
LIN {X 0,Y 272.682,Z 456.043,A -85,B 0,C 180,E1 16859.87,E2 16859.87} C_VEL
LIN {X 0,Y 280.623,Z 430.934,A -85,B 0,C 180,E1 16864.608,E2 16864.608} C_VEL
LIN {X 0,Y 288.768,Z 401.849,A -85,B 0,C 180,E1 16868.206,E2 16868.206} C_VEL
LIN {X 0,Y 294.466,Z 373.099,A -85,B 0,C 180,E1 16870.52,E2 16870.52} C_VEL
LIN {X 0,Y 287.061,Z 348.85,A -85,B 0,C 180,E1 16873.775,E2 16873.775} C_VEL
LIN {X 0,Y 273.819,Z 323.115,A -85,B 0,C 180,E1 16878.246,E2 16878.246} C_VEL
LIN {X 0,Y 264.129,Z 309.19,A -85,B 0,C 180,E1 16881.944,E2 16881.944} C_VEL
LIN {X 0,Y 260.929,Z 304.218,A -85,B 0,C 180,E1 16883.4,E2 16883.4} C_VEL
LIN {X 0,Y 257.842,Z 299.269,A -85,B 0,C 180,E1 16884.952,E2 16884.952} C_VEL
LIN {X 0,Y 257.729,Z 297.81,A -85,B 0,C 180,E1 16885.333,E2 16885.333} C_VEL
LIN {X 0,Y 257.923,Z 297.81,A -85,B 0,C 180,E1 16892.115,E2 16892.115} C_VEL
LIN {X 0,Y 258.383,Z 297.81,A -85,B 0,C 180,E1 16899.509,E2 16899.509} C_VEL
LIN {X 0,Y 258.879,Z 297.81,A -85,B 0,C 180,E1 16906.674,E2 16906.674} C_VEL
LIN {X 0,Y 256.455,Z 297.81,A -85,B 0,C 180,E1 16909.533,E2 16909.533} C_VEL
LIN {X 0,Y 251.582,Z 297.81,A -85,B 0,C 180,E1 16914.383,E2 16914.383} C_VEL
LIN {X 0,Y 251.965,Z 297.81,A -85,B 0,C 180,E1 16921.737,E2 16921.737} C_VEL
LIN {X 0,Y 251.955,Z 298.668,A -85,B 0,C 180,E1 16922.489,E2 16922.489} C_VEL
LIN {X 0,Y 254.902,Z 304.087,A -85,B 0,C 180,E1 16924.371,E2 16924.371} C_VEL
LIN {X 0,Y 256.727,Z 306.559,A -85,B 0,C 180,E1 16925.376,E2 16925.376} C_VEL
LIN {X 0,Y 265.264,Z 320.726,A -85,B 0,C 180,E1 16929.642,E2 16929.642} C_VEL
LIN {X 0,Y 273.598,Z 338.927,A -85,B 0,C 180,E1 16933.984,E2 16933.984} C_VEL
LIN {X 0,Y 279.101,Z 360.562,A -85,B 0,C 180,E1 16938.337,E2 16938.337} C_VEL
LIN {X 0,Y 280.254,Z 377.954,A -85,B 0,C 180,E1 16941.748,E2 16941.748} C_VEL
LIN {X 0,Y 272.753,Z 400.941,A -85,B 0,C 180,E1 16946.056,E2 16946.056} C_VEL
LIN {X 0,Y 266.082,Z 417.996,A -85,B 0,C 180,E1 16951.093,E2 16951.093} C_VEL
LIN {X 0,Y 261.291,Z 428.477,A -85,B 0,C 180,E1 16956.05,E2 16956.05} C_VEL
LIN {X 0,Y 258.357,Z 434.177,A -85,B 0,C 180,E1 16960.599,E2 16960.599} C_VEL
LIN {X 0,Y 256.412,Z 436.733,A -85,B 0,C 180,E1 16965.074,E2 16965.074} C_VEL
LIN {X 0,Y 255.391,Z 435.167,A -85,B 0,C 180,E1 16972.042,E2 16972.042} C_VEL
LIN {X 0,Y 256.542,Z 428.336,A -85,B 0,C 180,E1 16978.037,E2 16978.037} C_VEL
LIN {X 0,Y 259.143,Z 416.569,A -85,B 0,C 180,E1 16983.632,E2 16983.632} C_VEL
LIN {X 0,Y 263.124,Z 398.605,A -85,B 0,C 180,E1 16988.98,E2 16988.98} C_VEL
LIN {X 0,Y 267.024,Z 377.568,A -85,B 0,C 180,E1 16993.166,E2 16993.166} C_VEL
LIN {X 0,Y 265.648,Z 376.608,A -85,B 0,C 180,E1 16993.607,E2 16993.607} C_VEL
LIN {X 0,Y 262.58,Z 397.042,A -85,B 0,C 180,E1 16997.134,E2 16997.134} C_VEL
LIN {X 0,Y 259.269,Z 414.876,A -85,B 0,C 180,E1 17001.929,E2 17001.929} C_VEL
LIN {X 0,Y 256.77,Z 427.409,A -85,B 0,C 180,E1 17007.475,E2 17007.475} C_VEL
LIN {X 0,Y 255.49,Z 434.273,A -85,B 0,C 180,E1 17013.387,E2 17013.387} C_VEL
LIN {X 0,Y 255.428,Z 435.725,A -85,B 0,C 180,E1 17016.787,E2 17016.787} C_VEL
LIN {X 0,Y 256.53,Z 434.607,A -85,B 0,C 180,E1 17021.882,E2 17021.882} C_VEL
LIN {X 0,Y 259.253,Z 428.154,A -85,B 0,C 180,E1 17027.794,E2 17027.794} C_VEL
LIN {X 0,Y 263.179,Z 416.328,A -85,B 0,C 180,E1 17033.163,E2 17033.163} C_VEL
LIN {X 0,Y 267.872,Z 399.843,A -85,B 0,C 180,E1 17037.695,E2 17037.695} C_VEL
LIN {X 0,Y 272.31,Z 380.14,A -85,B 0,C 180,E1 17041.175,E2 17041.175} C_VEL
LIN {X 0,Y 274.124,Z 364.271,A -85,B 0,C 180,E1 17043.186,E2 17043.186} C_VEL
LIN {X 0,Y 268.954,Z 341.126,A -85,B 0,C 180,E1 17046.035,E2 17046.035} C_VEL
LIN {X 0,Y 257.613,Z 314.68,A -85,B 0,C 180,E1 17048.89,E2 17048.89} C_VEL
LIN {X 0,Y 249.555,Z 297.81,A -85,B 0,C 180,E1 17050.955,E2 17050.955} C_VEL
LIN {X 0,Y 249.455,Z 297.81,A -85,B 0,C 180,E1 17058.256,E2 17058.256} C_VEL
LIN {X 0,Y 249.821,Z 297.81,A -85,B 0,C 180,E1 17067.743,E2 17067.743} C_VEL
LIN {X 0,Y 250.166,Z 297.81,A -85,B 0,C 180,E1 17074.999,E2 17074.999} C_VEL
LIN {X 0,Y 250.687,Z 297.81,A -85,B 0,C 180,E1 17082.461,E2 17082.461} C_VEL
LIN {X 0,Y 251.229,Z 297.81,A -85,B 0,C 180,E1 17089.597,E2 17089.597} C_VEL
LIN {X 0,Y 251.977,Z 297.81,A -85,B 0,C 180,E1 17096.545,E2 17096.545} C_VEL
LIN {X 0,Y 252.309,Z 297.81,A -85,B 0,C 180,E1 17099.979,E2 17099.979} C_VEL
LIN {X 0,Y 251.627,Z 297.81,A -85,B 0,C 180,E1 17106.867,E2 17106.867} C_VEL
LIN {X 0,Y 250.844,Z 297.81,A -85,B 0,C 180,E1 17115.736,E2 17115.736} C_VEL
LIN {X 0,Y 250.477,Z 297.81,A -85,B 0,C 180,E1 17121.168,E2 17121.168} C_VEL
LIN {X 0,Y 249.968,Z 297.81,A -85,B 0,C 180,E1 17128.854,E2 17128.854} C_VEL
LIN {X 0,Y 249.579,Z 297.81,A -85,B 0,C 180,E1 17137.176,E2 17137.176} C_VEL
LIN {X 0,Y 249.718,Z 298.331,A -85,B 0,C 180,E1 17145.351,E2 17145.351} C_VEL
LIN {X 0,Y 270.241,Z 347.016,A -85,B 0,C 180,E1 17149.661,E2 17149.661} C_VEL
LIN {X 0,Y 277.467,Z 373.409,A -85,B 0,C 180,E1 17152.022,E2 17152.022} C_VEL
LIN {X 0,Y 272.15,Z 405.115,A -85,B 0,C 180,E1 17154.638,E2 17154.638} C_VEL
LIN {X 0,Y 266.09,Z 433.259,A -85,B 0,C 180,E1 17158.362,E2 17158.362} C_VEL
LIN {X 0,Y 260.259,Z 458.043,A -85,B 0,C 180,E1 17163.277,E2 17163.277} C_VEL
LIN {X 0,Y 255.847,Z 478.503,A -85,B 0,C 180,E1 17169.274,E2 17169.274} C_VEL
LIN {X 0,Y 253.904,Z 494.229,A -85,B 0,C 180,E1 17176.247,E2 17176.247} C_VEL
LIN {X 0,Y 254.321,Z 503.655,A -85,B 0,C 180,E1 17183.184,E2 17183.184} C_VEL
LIN {X 0,Y 254.767,Z 506.138,A -85,B 0,C 180,E1 17186.603,E2 17186.603} C_VEL
LIN {X 0,Y 255.06,Z 507.317,A -85,B 0,C 180,E1 17189.999,E2 17189.999} C_VEL
LIN {X 0,Y 254.605,Z 507.012,A -85,B 0,C 180,E1 17193.397,E2 17193.397} C_VEL
LIN {X 0,Y 253.663,Z 502.576,A -85,B 0,C 180,E1 17200.279,E2 17200.279} C_VEL
LIN {X 0,Y 254.712,Z 491.593,A -85,B 0,C 180,E1 17208.036,E2 17208.036} C_VEL
LIN {X 0,Y 259.086,Z 475.046,A -85,B 0,C 180,E1 17215.124,E2 17215.124} C_VEL
LIN {X 0,Y 266.462,Z 453.309,A -85,B 0,C 180,E1 17221.219,E2 17221.219} C_VEL
LIN {X 0,Y 275.188,Z 426.903,A -85,B 0,C 180,E1 17226.119,E2 17226.119} C_VEL
LIN {X 0,Y 283.491,Z 398.236,A -85,B 0,C 180,E1 17229.543,E2 17229.543} C_VEL
LIN {X 0,Y 288.172,Z 375.241,A -85,B 0,C 180,E1 17231.428,E2 17231.428} C_VEL
LIN {X 0,Y 281.261,Z 351.829,A -85,B 0,C 180,E1 17234.817,E2 17234.817} C_VEL
LIN {X 0,Y 269.887,Z 328.864,A -85,B 0,C 180,E1 17239.089,E2 17239.089} C_VEL
LIN {X 0,Y 258.056,Z 311.01,A -85,B 0,C 180,E1 17244.11,E2 17244.11} C_VEL
LIN {X 0,Y 253.658,Z 304.603,A -85,B 0,C 180,E1 17246.448,E2 17246.448} C_VEL
LIN {X 0,Y 250.095,Z 299.707,A -85,B 0,C 180,E1 17248.615,E2 17248.615} C_VEL
LIN {X 0,Y 249.836,Z 297.81,A -85,B 0,C 180,E1 17249.134,E2 17249.134} C_VEL
LIN {X 0,Y 250.143,Z 297.81,A -85,B 0,C 180,E1 17255.045,E2 17255.045} C_VEL
LIN {X 0,Y 250.631,Z 297.81,A -85,B 0,C 180,E1 17262.502,E2 17262.502} C_VEL
LIN {X 0,Y 251.186,Z 297.81,A -85,B 0,C 180,E1 17269.639,E2 17269.639} C_VEL
LIN {X 0,Y 251.582,Z 297.81,A -85,B 0,C 180,E1 17274.383,E2 17274.383} C_VEL
LIN {X 0,Y 248.066,Z 299.41,A -85,B 0,C 180,E1 17277,E2 17277} C_VEL
LIN {X 0,Y 245.798,Z 302.437,A -85,B 0,C 180,E1 17279.245,E2 17279.245} C_VEL
LIN {X 0,Y 246.091,Z 302.917,A -85,B 0,C 180,E1 17279.562,E2 17279.562} C_VEL
LIN {X 0,Y 249.379,Z 306.328,A -85,B 0,C 180,E1 17281.864,E2 17281.864} C_VEL
LIN {X 0,Y 257.93,Z 320.129,A -85,B 0,C 180,E1 17286.97,E2 17286.97} C_VEL
LIN {X 0,Y 266.48,Z 337.952,A -85,B 0,C 180,E1 17291.87,E2 17291.87} C_VEL
LIN {X 0,Y 272.44,Z 360.058,A -85,B 0,C 180,E1 17296.719,E2 17296.719} C_VEL
LIN {X 0,Y 273.881,Z 379.447,A -85,B 0,C 180,E1 17300.762,E2 17300.762} C_VEL
LIN {X 0,Y 266.418,Z 401.543,A -85,B 0,C 180,E1 17305.011,E2 17305.011} C_VEL
LIN {X 0,Y 259.288,Z 418.747,A -85,B 0,C 180,E1 17310.152,E2 17310.152} C_VEL
LIN {X 0,Y 253.929,Z 429.733,A -85,B 0,C 180,E1 17315.459,E2 17315.459} C_VEL
LIN {X 0,Y 249.974,Z 436.492,A -85,B 0,C 180,E1 17321.638,E2 17321.638} C_VEL
LIN {X 0,Y 247.865,Z 437.998,A -85,B 0,C 180,E1 17327.959,E2 17327.959} C_VEL
LIN {X 0,Y 247.838,Z 434.216,A -85,B 0,C 180,E1 17334.396,E2 17334.396} C_VEL
LIN {X 0,Y 249.597,Z 425.624,A -85,B 0,C 180,E1 17340.34,E2 17340.34} C_VEL
LIN {X 0,Y 253.041,Z 410.703,A -85,B 0,C 180,E1 17346.349,E2 17346.349} C_VEL
LIN {X 0,Y 257.517,Z 391.062,A -85,B 0,C 180,E1 17351.387,E2 17351.387} C_VEL
LIN {X 0,Y 259.276,Z 382.311,A -85,B 0,C 180,E1 17353.083,E2 17353.083} C_VEL
LIN {X 0,Y 257.73,Z 381.799,A -85,B 0,C 180,E1 17353.635,E2 17353.635} C_VEL
LIN {X 0,Y 254.325,Z 402.198,A -85,B 0,C 180,E1 17357.581,E2 17357.581} C_VEL
LIN {X 0,Y 251.027,Z 418.779,A -85,B 0,C 180,E1 17362.619,E2 17362.619} C_VEL
LIN {X 0,Y 248.671,Z 429.976,A -85,B 0,C 180,E1 17368.262,E2 17368.262} C_VEL
LIN {X 0,Y 247.651,Z 435.428,A -85,B 0,C 180,E1 17373.494,E2 17373.494} C_VEL
LIN {X 0,Y 247.616,Z 436.82,A -85,B 0,C 180,E1 17377.002,E2 17377.002} C_VEL
LIN {X 0,Y 248.822,Z 435.618,A -85,B 0,C 180,E1 17382.256,E2 17382.256} C_VEL
LIN {X 0,Y 251.737,Z 429.064,A -85,B 0,C 180,E1 17388.344,E2 17388.344} C_VEL
LIN {X 0,Y 255.952,Z 417.117,A -85,B 0,C 180,E1 17393.857,E2 17393.857} C_VEL
LIN {X 0,Y 260.856,Z 400.536,A -85,B 0,C 180,E1 17398.488,E2 17398.488} C_VEL
LIN {X 0,Y 265.774,Z 379.407,A -85,B 0,C 180,E1 17402.21,E2 17402.21} C_VEL
LIN {X 0,Y 267.266,Z 366.17,A -85,B 0,C 180,E1 17403.93,E2 17403.93} C_VEL
LIN {X 0,Y 262.121,Z 342.851,A -85,B 0,C 180,E1 17406.951,E2 17406.951} C_VEL
LIN {X 0,Y 251.024,Z 316.957,A -85,B 0,C 180,E1 17409.925,E2 17409.925} C_VEL
LIN {X 0,Y 241.587,Z 298.603,A -85,B 0,C 180,E1 17412.352,E2 17412.352} C_VEL
LIN {X 0,Y 241.519,Z 297.81,A -85,B 0,C 180,E1 17418.57,E2 17418.57} C_VEL
LIN {X 0,Y 241.635,Z 297.81,A -85,B 0,C 180,E1 17425.774,E2 17425.774} C_VEL
LIN {X 0,Y 242.152,Z 297.81,A -85,B 0,C 180,E1 17434.112,E2 17434.112} C_VEL
LIN {X 0,Y 242.674,Z 297.81,A -85,B 0,C 180,E1 17441.862,E2 17441.862} C_VEL
LIN {X 0,Y 243.257,Z 297.81,A -85,B 0,C 180,E1 17449.252,E2 17449.252} C_VEL
LIN {X 0,Y 244.038,Z 297.81,A -85,B 0,C 180,E1 17456.433,E2 17456.433} C_VEL
LIN {X 0,Y 244.398,Z 297.81,A -85,B 0,C 180,E1 17459.978,E2 17459.978} C_VEL
LIN {X 0,Y 243.6,Z 297.81,A -85,B 0,C 180,E1 17467.629,E2 17467.629} C_VEL
LIN {X 0,Y 243.063,Z 297.81,A -85,B 0,C 180,E1 17474.356,E2 17474.356} C_VEL
LIN {X 0,Y 242.459,Z 297.81,A -85,B 0,C 180,E1 17481.904,E2 17481.904} C_VEL
LIN {X 0,Y 241.952,Z 297.81,A -85,B 0,C 180,E1 17489.905,E2 17489.905} C_VEL
LIN {X 0,Y 241.576,Z 297.81,A -85,B 0,C 180,E1 17498.629,E2 17498.629} C_VEL
LIN {X 0,Y 241.746,Z 298.484,A -85,B 0,C 180,E1 17504.167,E2 17504.167} C_VEL
LIN {X 0,Y 262.308,Z 346.434,A -85,B 0,C 180,E1 17508.687,E2 17508.687} C_VEL
LIN {X 0,Y 270.283,Z 374.252,A -85,B 0,C 180,E1 17511.344,E2 17511.344} C_VEL
LIN {X 0,Y 264.819,Z 405.282,A -85,B 0,C 180,E1 17514.01,E2 17514.01} C_VEL
LIN {X 0,Y 258.378,Z 433.979,A -85,B 0,C 180,E1 17517.979,E2 17517.979} C_VEL
LIN {X 0,Y 252.482,Z 458.08,A -85,B 0,C 180,E1 17522.983,E2 17522.983} C_VEL
LIN {X 0,Y 248.018,Z 478.054,A -85,B 0,C 180,E1 17529.073,E2 17529.073} C_VEL
LIN {X 0,Y 246.094,Z 492.761,A -85,B 0,C 180,E1 17535.801,E2 17535.801} C_VEL
LIN {X 0,Y 246.167,Z 500.843,A -85,B 0,C 180,E1 17541.184,E2 17541.184} C_VEL
LIN {X 0,Y 246.917,Z 504.942,A -85,B 0,C 180,E1 17546.495,E2 17546.495} C_VEL
LIN {X 0,Y 247.23,Z 506.165,A -85,B 0,C 180,E1 17549.999,E2 17549.999} C_VEL
LIN {X 0,Y 246.74,Z 505.9,A -85,B 0,C 180,E1 17553.505,E2 17553.505} C_VEL
LIN {X 0,Y 245.768,Z 501.293,A -85,B 0,C 180,E1 17560.876,E2 17560.876} C_VEL
LIN {X 0,Y 246.989,Z 490.678,A -85,B 0,C 180,E1 17568.621,E2 17568.621} C_VEL
LIN {X 0,Y 251.397,Z 475.337,A -85,B 0,C 180,E1 17575.515,E2 17575.515} C_VEL
LIN {X 0,Y 258.841,Z 454.75,A -85,B 0,C 180,E1 17581.646,E2 17581.646} C_VEL
LIN {X 0,Y 267.519,Z 430.08,A -85,B 0,C 180,E1 17586.569,E2 17586.569} C_VEL
LIN {X 0,Y 276.616,Z 401.132,A -85,B 0,C 180,E1 17590.289,E2 17590.289} C_VEL
LIN {X 0,Y 282.147,Z 378.554,A -85,B 0,C 180,E1 17592.203,E2 17592.203} C_VEL
LIN {X 0,Y 275.753,Z 355.317,A -85,B 0,C 180,E1 17595.827,E2 17595.827} C_VEL
LIN {X 0,Y 265.883,Z 334.448,A -85,B 0,C 180,E1 17599.983,E2 17599.983} C_VEL
LIN {X 0,Y 255.269,Z 317.823,A -85,B 0,C 180,E1 17604.806,E2 17604.806} C_VEL
LIN {X 0,Y 250.621,Z 311.286,A -85,B 0,C 180,E1 17607.422,E2 17607.422} C_VEL
LIN {X 0,Y 246.601,Z 305.004,A -85,B 0,C 180,E1 17610.21,E2 17610.21} C_VEL
LIN {X 0,Y 242.459,Z 300.25,A -85,B 0,C 180,E1 17613.7,E2 17613.7} C_VEL
LIN {X 0,Y 242.178,Z 297.81,A -85,B 0,C 180,E1 17614.412,E2 17614.412} C_VEL
LIN {X 0,Y 242.62,Z 297.81,A -85,B 0,C 180,E1 17621.905,E2 17621.905} C_VEL
LIN {X 0,Y 243.213,Z 297.81,A -85,B 0,C 180,E1 17629.295,E2 17629.295} C_VEL
LIN {X 0,Y 244.068,Z 298.327,A -85,B 0,C 180,E1 17637.586,E2 17637.586} C_VEL
LIN {X 0,Y 246.091,Z 302.917,A -85,B 0,C 180,E1 17639.562,E2 17639.562} C_VEL
LIN {X 0,Y 247.682,Z 308.572,A -85,B 0,C 180,E1 17641.124,E2 17641.124} C_VEL
LIN {X 0,Y 249.569,Z 317.895,A -85,B 0,C 180,E1 17643.085,E2 17643.085} C_VEL
LIN {X 0,Y 250.286,Z 318.727,A -85,B 0,C 180,E1 17643.522,E2 17643.522} C_VEL
LIN {X 0,Y 259.031,Z 336.267,A -85,B 0,C 180,E1 17649.248,E2 17649.248} C_VEL
LIN {X 0,Y 265.171,Z 355.752,A -85,B 0,C 180,E1 17654.101,E2 17654.101} C_VEL
LIN {X 0,Y 267.599,Z 377.462,A -85,B 0,C 180,E1 17658.927,E2 17658.927} C_VEL
LIN {X 0,Y 266.154,Z 386.3,A -85,B 0,C 180,E1 17660.679,E2 17660.679} C_VEL
LIN {X 0,Y 258.405,Z 406.476,A -85,B 0,C 180,E1 17664.994,E2 17664.994} C_VEL
LIN {X 0,Y 251.091,Z 422.453,A -85,B 0,C 180,E1 17670.349,E2 17670.349} C_VEL
LIN {X 0,Y 245.049,Z 433.683,A -85,B 0,C 180,E1 17676.821,E2 17676.821} C_VEL
LIN {X 0,Y 241.316,Z 438.748,A -85,B 0,C 180,E1 17683.493,E2 17683.493} C_VEL
LIN {X 0,Y 239.875,Z 438.788,A -85,B 0,C 180,E1 17689.052,E2 17689.052} C_VEL
LIN {X 0,Y 240.223,Z 434.057,A -85,B 0,C 180,E1 17695.575,E2 17695.575} C_VEL
LIN {X 0,Y 242.508,Z 423.681,A -85,B 0,C 180,E1 17702.042,E2 17702.042} C_VEL
LIN {X 0,Y 246.504,Z 407.168,A -85,B 0,C 180,E1 17708.147,E2 17708.147} C_VEL
LIN {X 0,Y 251.18,Z 386.977,A -85,B 0,C 180,E1 17712.971,E2 17712.971} C_VEL
LIN {X 0,Y 249.861,Z 386.139,A -85,B 0,C 180,E1 17713.556,E2 17713.556} C_VEL
LIN {X 0,Y 246.065,Z 407.005,A -85,B 0,C 180,E1 17718.056,E2 17718.056} C_VEL
LIN {X 0,Y 242.799,Z 422.32,A -85,B 0,C 180,E1 17723.309,E2 17723.309} C_VEL
LIN {X 0,Y 240.599,Z 432.394,A -85,B 0,C 180,E1 17729.103,E2 17729.103} C_VEL
LIN {X 0,Y 239.829,Z 436.581,A -85,B 0,C 180,E1 17733.608,E2 17733.608} C_VEL
LIN {X 0,Y 239.807,Z 437.914,A -85,B 0,C 180,E1 17737.231,E2 17737.231} C_VEL
LIN {X 0,Y 241.143,Z 436.628,A -85,B 0,C 180,E1 17742.652,E2 17742.652} C_VEL
LIN {X 0,Y 244.246,Z 429.967,A -85,B 0,C 180,E1 17748.928,E2 17748.928} C_VEL
LIN {X 0,Y 248.829,Z 417.694,A -85,B 0,C 180,E1 17754.671,E2 17754.671} C_VEL
LIN {X 0,Y 254.217,Z 400.053,A -85,B 0,C 180,E1 17759.594,E2 17759.594} C_VEL
LIN {X 0,Y 259.35,Z 378.598,A -85,B 0,C 180,E1 17763.301,E2 17763.301} C_VEL
LIN {X 0,Y 260.213,Z 366.365,A -85,B 0,C 180,E1 17764.965,E2 17764.965} C_VEL
LIN {X 0,Y 254.942,Z 343.146,A -85,B 0,C 180,E1 17768.089,E2 17768.089} C_VEL
LIN {X 0,Y 242.269,Z 315.088,A -85,B 0,C 180,E1 17771.596,E2 17771.596} C_VEL
LIN {X 0,Y 233.687,Z 298.777,A -85,B 0,C 180,E1 17773.983,E2 17773.983} C_VEL
LIN {X 0,Y 233.599,Z 297.81,A -85,B 0,C 180,E1 17774.272,E2 17774.272} C_VEL
LIN {X 0,Y 233.606,Z 297.81,A -85,B 0,C 180,E1 17780.82,E2 17780.82} C_VEL
LIN {X 0,Y 233.802,Z 297.81,A -85,B 0,C 180,E1 17788.885,E2 17788.885} C_VEL
LIN {X 0,Y 234.359,Z 297.81,A -85,B 0,C 180,E1 17797.248,E2 17797.248} C_VEL
LIN {X 0,Y 234.969,Z 297.81,A -85,B 0,C 180,E1 17805.09,E2 17805.09} C_VEL
LIN {X 0,Y 235.685,Z 297.81,A -85,B 0,C 180,E1 17813.47,E2 17813.47} C_VEL
LIN {X 0,Y 236.495,Z 297.81,A -85,B 0,C 180,E1 17819.977,E2 17819.977} C_VEL
LIN {X 0,Y 235.751,Z 297.81,A -85,B 0,C 180,E1 17827.332,E2 17827.332} C_VEL
LIN {X 0,Y 234.94,Z 297.81,A -85,B 0,C 180,E1 17835.538,E2 17835.538} C_VEL
LIN {X 0,Y 234.26,Z 297.81,A -85,B 0,C 180,E1 17845.6,E2 17845.6} C_VEL
LIN {X 0,Y 233.71,Z 297.81,A -85,B 0,C 180,E1 17855.501,E2 17855.501} C_VEL
LIN {X 0,Y 233.689,Z 297.81,A -85,B 0,C 180,E1 17862.796,E2 17862.796} C_VEL
LIN {X 0,Y 254.091,Z 345.192,A -85,B 0,C 180,E1 17867.586,E2 17867.586} C_VEL
LIN {X 0,Y 263.036,Z 374.816,A -85,B 0,C 180,E1 17870.598,E2 17870.598} C_VEL
LIN {X 0,Y 257.475,Z 405.669,A -85,B 0,C 180,E1 17873.372,E2 17873.372} C_VEL
LIN {X 0,Y 250.845,Z 434.016,A -85,B 0,C 180,E1 17877.45,E2 17877.45} C_VEL
LIN {X 0,Y 244.711,Z 458.033,A -85,B 0,C 180,E1 17882.652,E2 17882.652} C_VEL
LIN {X 0,Y 240.053,Z 478.198,A -85,B 0,C 180,E1 17889.129,E2 17889.129} C_VEL
LIN {X 0,Y 238.105,Z 494.831,A -85,B 0,C 180,E1 17897.183,E2 17897.183} C_VEL
LIN {X 0,Y 238.502,Z 501.563,A -85,B 0,C 180,E1 17902.729,E2 17902.729} C_VEL
LIN {X 0,Y 239.414,Z 504.996,A -85,B 0,C 180,E1 17909.999,E2 17909.999} C_VEL
LIN {X 0,Y 238.855,Z 504.784,A -85,B 0,C 180,E1 17913.621,E2 17913.621} C_VEL
LIN {X 0,Y 237.879,Z 500.552,A -85,B 0,C 180,E1 17920.97,E2 17920.97} C_VEL
LIN {X 0,Y 239.406,Z 489.474,A -85,B 0,C 180,E1 17929.422,E2 17929.422} C_VEL
LIN {X 0,Y 244.734,Z 472.919,A -85,B 0,C 180,E1 17936.96,E2 17936.96} C_VEL
LIN {X 0,Y 253.142,Z 451.234,A -85,B 0,C 180,E1 17943.341,E2 17943.341} C_VEL
LIN {X 0,Y 262.936,Z 425.048,A -85,B 0,C 180,E1 17948.354,E2 17948.354} C_VEL
LIN {X 0,Y 271.762,Z 397.219,A -85,B 0,C 180,E1 17951.782,E2 17951.782} C_VEL
LIN {X 0,Y 275.802,Z 379.656,A -85,B 0,C 180,E1 17953.338,E2 17953.338} C_VEL
LIN {X 0,Y 269.389,Z 356.172,A -85,B 0,C 180,E1 17957.341,E2 17957.341} C_VEL
LIN {X 0,Y 259.753,Z 336.011,A -85,B 0,C 180,E1 17961.91,E2 17961.91} C_VEL
LIN {X 0,Y 249.126,Z 319.099,A -85,B 0,C 180,E1 17967.562,E2 17967.562} C_VEL
LIN {X 0,Y 244.219,Z 312.173,A -85,B 0,C 180,E1 17971.02,E2 17971.02} C_VEL
LIN {X 0,Y 240.35,Z 306.672,A -85,B 0,C 180,E1 17974.67,E2 17974.67} C_VEL
LIN {X 0,Y 238.927,Z 304.98,A -85,B 0,C 180,E1 17976.418,E2 17976.418} C_VEL
LIN {X 0,Y 235.661,Z 301.136,A -85,B 0,C 180,E1 17985.183,E2 17985.183} C_VEL
LIN {X 0,Y 239.618,Z 304.593,A -85,B 0,C 180,E1 17994.602,E2 17994.602} C_VEL
LIN {X 0,Y 242.049,Z 306.313,A -85,B 0,C 180,E1 17997.07,E2 17997.07} C_VEL
LIN {X 0,Y 247.438,Z 314.637,A -85,B 0,C 180,E1 18001.606,E2 18001.606} C_VEL
LIN {X 0,Y 250.286,Z 318.727,A -85,B 0,C 180,E1 18003.522,E2 18003.522} C_VEL
LIN {X 0,Y 253.004,Z 324.703,A -85,B 0,C 180,E1 18005.443,E2 18005.443} C_VEL
LIN {X 0,Y 255.119,Z 343.129,A -85,B 0,C 180,E1 18008.828,E2 18008.828} C_VEL
LIN {X 0,Y 255.364,Z 343.799,A -85,B 0,C 180,E1 18009.028,E2 18009.028} C_VEL
LIN {X 0,Y 260.173,Z 362.587,A -85,B 0,C 180,E1 18013.907,E2 18013.907} C_VEL
LIN {X 0,Y 261.271,Z 382.401,A -85,B 0,C 180,E1 18018.544,E2 18018.544} C_VEL
LIN {X 0,Y 256.686,Z 396.668,A -85,B 0,C 180,E1 18021.345,E2 18021.345} C_VEL
LIN {X 0,Y 248.416,Z 415.275,A -85,B 0,C 180,E1 18026.284,E2 18026.284} C_VEL
LIN {X 0,Y 241.38,Z 428.732,A -85,B 0,C 180,E1 18032.001,E2 18032.001} C_VEL
LIN {X 0,Y 236.346,Z 436.813,A -85,B 0,C 180,E1 18038.044,E2 18038.044} C_VEL
LIN {X 0,Y 232.789,Z 440.381,A -85,B 0,C 180,E1 18045.518,E2 18045.518} C_VEL
LIN {X 0,Y 231.926,Z 438.715,A -85,B 0,C 180,E1 18051.37,E2 18051.37} C_VEL
LIN {X 0,Y 232.841,Z 432.876,A -85,B 0,C 180,E1 18057.451,E2 18057.451} C_VEL
LIN {X 0,Y 235.565,Z 421.464,A -85,B 0,C 180,E1 18063.799,E2 18063.799} C_VEL
LIN {X 0,Y 239.966,Z 403.959,A -85,B 0,C 180,E1 18069.814,E2 18069.814} C_VEL
LIN {X 0,Y 243.006,Z 391.406,A -85,B 0,C 180,E1 18072.846,E2 18072.846} C_VEL
LIN {X 0,Y 241.994,Z 390.202,A -85,B 0,C 180,E1 18073.472,E2 18073.472} C_VEL
LIN {X 0,Y 238.128,Z 409.986,A -85,B 0,C 180,E1 18078.116,E2 18078.116} C_VEL
LIN {X 0,Y 234.821,Z 424.611,A -85,B 0,C 180,E1 18083.544,E2 18083.544} C_VEL
LIN {X 0,Y 232.563,Z 434.671,A -85,B 0,C 180,E1 18090.001,E2 18090.001} C_VEL
LIN {X 0,Y 231.989,Z 437.737,A -85,B 0,C 180,E1 18093.731,E2 18093.731} C_VEL
LIN {X 0,Y 232.003,Z 439.009,A -85,B 0,C 180,E1 18097.476,E2 18097.476} C_VEL
LIN {X 0,Y 233.448,Z 437.68,A -85,B 0,C 180,E1 18103.008,E2 18103.008} C_VEL
LIN {X 0,Y 236.786,Z 430.869,A -85,B 0,C 180,E1 18109.548,E2 18109.548} C_VEL
LIN {X 0,Y 241.661,Z 418.47,A -85,B 0,C 180,E1 18115.454,E2 18115.454} C_VEL
LIN {X 0,Y 247.244,Z 401.035,A -85,B 0,C 180,E1 18120.416,E2 18120.416} C_VEL
LIN {X 0,Y 252.728,Z 379.079,A -85,B 0,C 180,E1 18124.267,E2 18124.267} C_VEL
LIN {X 0,Y 253.481,Z 368.687,A -85,B 0,C 180,E1 18125.74,E2 18125.74} C_VEL
LIN {X 0,Y 248.458,Z 345.483,A -85,B 0,C 180,E1 18129.034,E2 18129.034} C_VEL
LIN {X 0,Y 236.201,Z 318.16,A -85,B 0,C 180,E1 18132.683,E2 18132.683} C_VEL
LIN {X 0,Y 225.635,Z 298.236,A -85,B 0,C 180,E1 18135.845,E2 18135.845} C_VEL
LIN {X 0,Y 225.647,Z 297.81,A -85,B 0,C 180,E1 18143.37,E2 18143.37} C_VEL
LIN {X 0,Y 226.026,Z 297.81,A -85,B 0,C 180,E1 18152.111,E2 18152.111} C_VEL
LIN {X 0,Y 226.645,Z 297.81,A -85,B 0,C 180,E1 18160.529,E2 18160.529} C_VEL
LIN {X 0,Y 227.289,Z 297.81,A -85,B 0,C 180,E1 18168.487,E2 18168.487} C_VEL
LIN {X 0,Y 228.153,Z 297.81,A -85,B 0,C 180,E1 18176.184,E2 18176.184} C_VEL
LIN {X 0,Y 228.582,Z 297.81,A -85,B 0,C 180,E1 18179.976,E2 18179.976} C_VEL
LIN {X 0,Y 227.783,Z 297.81,A -85,B 0,C 180,E1 18187.59,E2 18187.59} C_VEL
LIN {X 0,Y 227.059,Z 297.81,A -85,B 0,C 180,E1 18195.392,E2 18195.392} C_VEL
LIN {X 0,Y 226.419,Z 297.81,A -85,B 0,C 180,E1 18203.545,E2 18203.545} C_VEL
LIN {X 0,Y 225.876,Z 297.81,A -85,B 0,C 180,E1 18212.28,E2 18212.28} C_VEL
LIN {X 0,Y 225.788,Z 297.81,A -85,B 0,C 180,E1 18221.451,E2 18221.451} C_VEL
LIN {X 0,Y 246.569,Z 345.404,A -85,B 0,C 180,E1 18226.584,E2 18226.584} C_VEL
LIN {X 0,Y 255.772,Z 376.271,A -85,B 0,C 180,E1 18229.906,E2 18229.906} C_VEL
LIN {X 0,Y 249.888,Z 407.16,A -85,B 0,C 180,E1 18232.851,E2 18232.851} C_VEL
LIN {X 0,Y 243.199,Z 434.487,A -85,B 0,C 180,E1 18236.986,E2 18236.986} C_VEL
LIN {X 0,Y 236.781,Z 458.613,A -85,B 0,C 180,E1 18242.48,E2 18242.48} C_VEL
LIN {X 0,Y 232.153,Z 478.003,A -85,B 0,C 180,E1 18249.052,E2 18249.052} C_VEL
LIN {X 0,Y 230.244,Z 493.844,A -85,B 0,C 180,E1 18256.738,E2 18256.738} C_VEL
LIN {X 0,Y 230.607,Z 500.52,A -85,B 0,C 180,E1 18262.479,E2 18262.479} C_VEL
LIN {X 0,Y 231.583,Z 503.822,A -85,B 0,C 180,E1 18269.999,E2 18269.999} C_VEL
LIN {X 0,Y 230.983,Z 503.673,A -85,B 0,C 180,E1 18273.745,E2 18273.745} C_VEL
LIN {X 0,Y 229.991,Z 499.529,A -85,B 0,C 180,E1 18281.351,E2 18281.351} C_VEL
LIN {X 0,Y 231.521,Z 489.423,A -85,B 0,C 180,E1 18289.558,E2 18289.558} C_VEL
LIN {X 0,Y 236.966,Z 473.596,A -85,B 0,C 180,E1 18297.299,E2 18297.299} C_VEL
LIN {X 0,Y 245.663,Z 452.596,A -85,B 0,C 180,E1 18303.896,E2 18303.896} C_VEL
LIN {X 0,Y 255.364,Z 428.347,A -85,B 0,C 180,E1 18308.891,E2 18308.891} C_VEL
LIN {X 0,Y 265.333,Z 399.401,A -85,B 0,C 180,E1 18312.701,E2 18312.701} C_VEL
LIN {X 0,Y 269.718,Z 381.795,A -85,B 0,C 180,E1 18314.383,E2 18314.383} C_VEL
LIN {X 0,Y 263.895,Z 359.47,A -85,B 0,C 180,E1 18318.498,E2 18318.498} C_VEL
LIN {X 0,Y 255.507,Z 341.065,A -85,B 0,C 180,E1 18323.03,E2 18323.03} C_VEL
LIN {X 0,Y 246.542,Z 326.011,A -85,B 0,C 180,E1 18328.344,E2 18328.344} C_VEL
LIN {X 0,Y 241.864,Z 319.272,A -85,B 0,C 180,E1 18331.87,E2 18331.87} C_VEL
LIN {X 0,Y 238.43,Z 313.401,A -85,B 0,C 180,E1 18335.54,E2 18335.54} C_VEL
LIN {X 0,Y 234.446,Z 308.966,A -85,B 0,C 180,E1 18345.104,E2 18345.104} C_VEL
LIN {X 0,Y 237.911,Z 312.159,A -85,B 0,C 180,E1 18354.107,E2 18354.107} C_VEL
LIN {X 0,Y 240.192,Z 314.073,A -85,B 0,C 180,E1 18356.63,E2 18356.63} C_VEL
LIN {X 0,Y 245.08,Z 321.954,A -85,B 0,C 180,E1 18361.088,E2 18361.088} C_VEL
LIN {X 0,Y 251.526,Z 334.3,A -85,B 0,C 180,E1 18366.048,E2 18366.048} C_VEL
LIN {X 0,Y 255.364,Z 343.799,A -85,B 0,C 180,E1 18369.028,E2 18369.028} C_VEL
LIN {X 0,Y 256.615,Z 353.236,A -85,B 0,C 180,E1 18371.037,E2 18371.037} C_VEL
LIN {X 0,Y 255.042,Z 370.877,A -85,B 0,C 180,E1 18374.108,E2 18374.108} C_VEL
LIN {X 0,Y 254.91,Z 386.9,A -85,B 0,C 180,E1 18378.062,E2 18378.062} C_VEL
LIN {X 0,Y 245.704,Z 408.784,A -85,B 0,C 180,E1 18382.896,E2 18382.896} C_VEL
LIN {X 0,Y 237.366,Z 424.811,A -85,B 0,C 180,E1 18388.543,E2 18388.543} C_VEL
LIN {X 0,Y 231.12,Z 434.969,A -85,B 0,C 180,E1 18394.537,E2 18394.537} C_VEL
LIN {X 0,Y 226.389,Z 440.831,A -85,B 0,C 180,E1 18401.835,E2 18401.835} C_VEL
LIN {X 0,Y 224.159,Z 440.576,A -85,B 0,C 180,E1 18409.766,E2 18409.766} C_VEL
LIN {X 0,Y 224.652,Z 435.652,A -85,B 0,C 180,E1 18416.108,E2 18416.108} C_VEL
LIN {X 0,Y 227.459,Z 424.034,A -85,B 0,C 180,E1 18423.401,E2 18423.401} C_VEL
LIN {X 0,Y 231.762,Z 407.487,A -85,B 0,C 180,E1 18429.593,E2 18429.593} C_VEL
LIN {X 0,Y 234.811,Z 395.654,A -85,B 0,C 180,E1 18432.728,E2 18432.728} C_VEL
LIN {X 0,Y 234.097,Z 394.094,A -85,B 0,C 180,E1 18433.379,E2 18433.379} C_VEL
LIN {X 0,Y 230.2,Z 412.918,A -85,B 0,C 180,E1 18438.18,E2 18438.18} C_VEL
LIN {X 0,Y 226.622,Z 427.764,A -85,B 0,C 180,E1 18444.269,E2 18444.269} C_VEL
LIN {X 0,Y 224.737,Z 435.864,A -85,B 0,C 180,E1 18450.001,E2 18450.001} C_VEL
LIN {X 0,Y 224.161,Z 438.888,A -85,B 0,C 180,E1 18453.861,E2 18453.861} C_VEL
LIN {X 0,Y 224.216,Z 440.102,A -85,B 0,C 180,E1 18457.737,E2 18457.737} C_VEL
LIN {X 0,Y 225.642,Z 438.885,A -85,B 0,C 180,E1 18463.131,E2 18463.131} C_VEL
LIN {X 0,Y 229.345,Z 431.772,A -85,B 0,C 180,E1 18470.209,E2 18470.209} C_VEL
LIN {X 0,Y 234.418,Z 419.572,A -85,B 0,C 180,E1 18476.164,E2 18476.164} C_VEL
LIN {X 0,Y 240.231,Z 402.372,A -85,B 0,C 180,E1 18481.2,E2 18481.2} C_VEL
LIN {X 0,Y 246.06,Z 380.15,A -85,B 0,C 180,E1 18485.2,E2 18485.2} C_VEL
LIN {X 0,Y 246.749,Z 370.849,A -85,B 0,C 180,E1 18486.577,E2 18486.577} C_VEL
LIN {X 0,Y 242.182,Z 348.527,A -85,B 0,C 180,E1 18489.949,E2 18489.949} C_VEL
LIN {X 0,Y 231.132,Z 323.06,A -85,B 0,C 180,E1 18493.555,E2 18493.555} C_VEL
LIN {X 0,Y 217.723,Z 299.119,A -85,B 0,C 180,E1 18497.81,E2 18497.81} C_VEL
LIN {X 0,Y 217.619,Z 297.81,A -85,B 0,C 180,E1 18498.027,E2 18498.027} C_VEL
LIN {X 0,Y 217.739,Z 297.81,A -85,B 0,C 180,E1 18506.298,E2 18506.298} C_VEL
LIN {X 0,Y 218.278,Z 297.81,A -85,B 0,C 180,E1 18515.466,E2 18515.466} C_VEL
LIN {X 0,Y 219.091,Z 297.81,A -85,B 0,C 180,E1 18524.638,E2 18524.638} C_VEL
LIN {X 0,Y 219.812,Z 297.81,A -85,B 0,C 180,E1 18533.566,E2 18533.566} C_VEL
LIN {X 0,Y 220.667,Z 297.81,A -85,B 0,C 180,E1 18539.976,E2 18539.976} C_VEL
LIN {X 0,Y 219.812,Z 297.81,A -85,B 0,C 180,E1 18547.867,E2 18547.867} C_VEL
LIN {X 0,Y 219.055,Z 297.81,A -85,B 0,C 180,E1 18555.97,E2 18555.97} C_VEL
LIN {X 0,Y 218.329,Z 297.81,A -85,B 0,C 180,E1 18564.474,E2 18564.474} C_VEL
LIN {X 0,Y 217.776,Z 297.81,A -85,B 0,C 180,E1 18573.745,E2 18573.745} C_VEL
LIN {X 0,Y 217.818,Z 297.81,A -85,B 0,C 180,E1 18579.998,E2 18579.998} C_VEL
LIN {X 0,Y 238.744,Z 344.906,A -85,B 0,C 180,E1 18585.452,E2 18585.452} C_VEL
LIN {X 0,Y 248.026,Z 375.641,A -85,B 0,C 180,E1 18588.927,E2 18588.927} C_VEL
LIN {X 0,Y 247.307,Z 385.541,A -85,B 0,C 180,E1 18589.848,E2 18589.848} C_VEL
LIN {X 0,Y 240.795,Z 415.076,A -85,B 0,C 180,E1 18593.182,E2 18593.182} C_VEL
LIN {X 0,Y 233.403,Z 442.633,A -85,B 0,C 180,E1 18598.088,E2 18598.088} C_VEL
LIN {X 0,Y 227.332,Z 465.174,A -85,B 0,C 180,E1 18604.181,E2 18604.181} C_VEL
LIN {X 0,Y 223.035,Z 486.319,A -85,B 0,C 180,E1 18612.527,E2 18612.527} C_VEL
LIN {X 0,Y 222.411,Z 496.757,A -85,B 0,C 180,E1 18619.275,E2 18619.275} C_VEL
LIN {X 0,Y 223.325,Z 501.487,A -85,B 0,C 180,E1 18626.124,E2 18626.124} C_VEL
LIN {X 0,Y 223.767,Z 502.652,A -85,B 0,C 180,E1 18629.999,E2 18629.999} C_VEL
LIN {X 0,Y 223.097,Z 502.559,A -85,B 0,C 180,E1 18633.877,E2 18633.877} C_VEL
LIN {X 0,Y 222.1,Z 498.498,A -85,B 0,C 180,E1 18641.76,E2 18641.76} C_VEL
LIN {X 0,Y 224.097,Z 487.868,A -85,B 0,C 180,E1 18650.701,E2 18650.701} C_VEL
LIN {X 0,Y 230.479,Z 471.297,A -85,B 0,C 180,E1 18658.871,E2 18658.871} C_VEL
LIN {X 0,Y 240.085,Z 449.894,A -85,B 0,C 180,E1 18665.545,E2 18665.545} C_VEL
LIN {X 0,Y 250.656,Z 424.699,A -85,B 0,C 180,E1 18670.611,E2 18670.611} C_VEL
LIN {X 0,Y 260.574,Z 396.53,A -85,B 0,C 180,E1 18674.213,E2 18674.213} C_VEL
LIN {X 0,Y 263.657,Z 383.64,A -85,B 0,C 180,E1 18675.511,E2 18675.511} C_VEL
LIN {X 0,Y 258.082,Z 361.518,A -85,B 0,C 180,E1 18679.997,E2 18679.997} C_VEL
LIN {X 0,Y 250.322,Z 343.902,A -85,B 0,C 180,E1 18684.824,E2 18684.824} C_VEL
LIN {X 0,Y 242.904,Z 331.467,A -85,B 0,C 180,E1 18689.902,E2 18689.902} C_VEL
LIN {X 0,Y 239.811,Z 326.497,A -85,B 0,C 180,E1 18692.571,E2 18692.571} C_VEL
LIN {X 0,Y 236.029,Z 320.369,A -85,B 0,C 180,E1 18697.054,E2 18697.054} C_VEL
LIN {X 0,Y 233.261,Z 316.825,A -85,B 0,C 180,E1 18706.013,E2 18706.013} C_VEL
LIN {X 0,Y 238.177,Z 321.383,A -85,B 0,C 180,E1 18716.049,E2 18716.049} C_VEL
LIN {X 0,Y 242.623,Z 329.488,A -85,B 0,C 180,E1 18720.714,E2 18720.714} C_VEL
LIN {X 0,Y 248.093,Z 341.247,A -85,B 0,C 180,E1 18725.622,E2 18725.622} C_VEL
LIN {X 0,Y 253.499,Z 359.548,A -85,B 0,C 180,E1 18731.177,E2 18731.177} C_VEL
LIN {X 0,Y 255.042,Z 370.877,A -85,B 0,C 180,E1 18734.108,E2 18734.108} C_VEL
LIN {X 0,Y 253.27,Z 380.932,A -85,B 0,C 180,E1 18735.979,E2 18735.979} C_VEL
LIN {X 0,Y 245.209,Z 398.103,A -85,B 0,C 180,E1 18738.814,E2 18738.814} C_VEL
LIN {X 0,Y 235.554,Z 417.475,A -85,B 0,C 180,E1 18744.113,E2 18744.113} C_VEL
LIN {X 0,Y 227.266,Z 431.3,A -85,B 0,C 180,E1 18750.328,E2 18750.328} C_VEL
LIN {X 0,Y 221.419,Z 439.335,A -85,B 0,C 180,E1 18756.868,E2 18756.868} C_VEL
LIN {X 0,Y 217.632,Z 442.597,A -85,B 0,C 180,E1 18763.934,E2 18763.934} C_VEL
LIN {X 0,Y 216.281,Z 440.019,A -85,B 0,C 180,E1 18772.511,E2 18772.511} C_VEL
LIN {X 0,Y 218.021,Z 431.538,A -85,B 0,C 180,E1 18780.066,E2 18780.066} C_VEL
LIN {X 0,Y 221.786,Z 417.336,A -85,B 0,C 180,E1 18787.059,E2 18787.059} C_VEL
LIN {X 0,Y 226.613,Z 397.974,A -85,B 0,C 180,E1 18793.064,E2 18793.064} C_VEL
LIN {X 0,Y 221.288,Z 419.655,A -85,B 0,C 180,E1 18799.689,E2 18799.689} C_VEL
LIN {X 0,Y 218.033,Z 432.231,A -85,B 0,C 180,E1 18806.033,E2 18806.033} C_VEL
LIN {X 0,Y 216.55,Z 438.76,A -85,B 0,C 180,E1 18811.998,E2 18811.998} C_VEL
LIN {X 0,Y 216.422,Z 441.197,A -85,B 0,C 180,E1 18818.017,E2 18818.017} C_VEL
LIN {X 0,Y 218.39,Z 439.336,A -85,B 0,C 180,E1 18824.577,E2 18824.577} C_VEL
LIN {X 0,Y 221.958,Z 432.675,A -85,B 0,C 180,E1 18830.913,E2 18830.913} C_VEL
LIN {X 0,Y 227.486,Z 419.997,A -85,B 0,C 180,E1 18837.169,E2 18837.169} C_VEL
LIN {X 0,Y 233.718,Z 402.191,A -85,B 0,C 180,E1 18842.391,E2 18842.391} C_VEL
LIN {X 0,Y 239.627,Z 380.483,A -85,B 0,C 180,E1 18846.293,E2 18846.293} C_VEL
LIN {X 0,Y 239.666,Z 369.098,A -85,B 0,C 180,E1 18848.12,E2 18848.12} C_VEL
LIN {X 0,Y 234.313,Z 346.408,A -85,B 0,C 180,E1 18851.674,E2 18851.674} C_VEL
LIN {X 0,Y 221.061,Z 318.542,A -85,B 0,C 180,E1 18856.074,E2 18856.074} C_VEL
LIN {X 0,Y 209.825,Z 299.769,A -85,B 0,C 180,E1 18860.009,E2 18860.009} C_VEL
LIN {X 0,Y 209.579,Z 297.81,A -85,B 0,C 180,E1 18860.331,E2 18860.331} C_VEL
LIN {X 0,Y 209.922,Z 297.81,A -85,B 0,C 180,E1 18869.758,E2 18869.758} C_VEL
LIN {X 0,Y 210.566,Z 297.81,A -85,B 0,C 180,E1 18878.975,E2 18878.975} C_VEL
LIN {X 0,Y 211.347,Z 297.81,A -85,B 0,C 180,E1 18887.605,E2 18887.605} C_VEL
LIN {X 0,Y 212.289,Z 297.81,A -85,B 0,C 180,E1 18895.898,E2 18895.898} C_VEL
LIN {X 0,Y 212.753,Z 297.81,A -85,B 0,C 180,E1 18899.975,E2 18899.975} C_VEL
LIN {X 0,Y 211.859,Z 297.81,A -85,B 0,C 180,E1 18908.164,E2 18908.164} C_VEL
LIN {X 0,Y 211.017,Z 297.81,A -85,B 0,C 180,E1 18916.595,E2 18916.595} C_VEL
LIN {X 0,Y 210.314,Z 297.81,A -85,B 0,C 180,E1 18925.472,E2 18925.472} C_VEL
LIN {X 0,Y 209.749,Z 297.81,A -85,B 0,C 180,E1 18935.108,E2 18935.108} C_VEL
LIN {X 0,Y 209.925,Z 298.375,A -85,B 0,C 180,E1 18938.506,E2 18938.506} C_VEL
LIN {X 0,Y 230.977,Z 344.692,A -85,B 0,C 180,E1 18944.255,E2 18944.255} C_VEL
LIN {X 0,Y 240.483,Z 375.686,A -85,B 0,C 180,E1 18947.987,E2 18947.987} C_VEL
LIN {X 0,Y 241.041,Z 381.543,A -85,B 0,C 180,E1 18948.666,E2 18948.666} C_VEL
LIN {X 0,Y 234.338,Z 411.76,A -85,B 0,C 180,E1 18951.991,E2 18951.991} C_VEL
LIN {X 0,Y 226.801,Z 439.054,A -85,B 0,C 180,E1 18956.764,E2 18956.764} C_VEL
LIN {X 0,Y 220.326,Z 461.931,A -85,B 0,C 180,E1 18962.869,E2 18962.869} C_VEL
LIN {X 0,Y 215.837,Z 482.283,A -85,B 0,C 180,E1 18970.371,E2 18970.371} C_VEL
LIN {X 0,Y 214.489,Z 493.301,A -85,B 0,C 180,E1 18976.781,E2 18976.781} C_VEL
LIN {X 0,Y 214.797,Z 498.432,A -85,B 0,C 180,E1 18981.922,E2 18981.922} C_VEL
LIN {X 0,Y 215.933,Z 501.467,A -85,B 0,C 180,E1 18989.999,E2 18989.999} C_VEL
LIN {X 0,Y 215.215,Z 501.447,A -85,B 0,C 180,E1 18994.019,E2 18994.019} C_VEL
LIN {X 0,Y 214.226,Z 497.474,A -85,B 0,C 180,E1 19002.198,E2 19002.198} C_VEL
LIN {X 0,Y 216.533,Z 486.998,A -85,B 0,C 180,E1 19011.46,E2 19011.46} C_VEL
LIN {X 0,Y 223.447,Z 470.642,A -85,B 0,C 180,E1 19019.87,E2 19019.87} C_VEL
LIN {X 0,Y 233.579,Z 449.457,A -85,B 0,C 180,E1 19026.696,E2 19026.696} C_VEL
LIN {X 0,Y 244.656,Z 424.6,A -85,B 0,C 180,E1 19031.827,E2 19031.827} C_VEL
LIN {X 0,Y 255.367,Z 395.787,A -85,B 0,C 180,E1 19035.562,E2 19035.562} C_VEL
LIN {X 0,Y 257.858,Z 386.928,A -85,B 0,C 180,E1 19036.461,E2 19036.461} C_VEL
LIN {X 0,Y 252.838,Z 365.002,A -85,B 0,C 180,E1 19041.219,E2 19041.219} C_VEL
LIN {X 0,Y 245.552,Z 347.869,A -85,B 0,C 180,E1 19046.447,E2 19046.447} C_VEL
LIN {X 0,Y 238.533,Z 334.552,A -85,B 0,C 180,E1 19052.412,E2 19052.412} C_VEL
LIN {X 0,Y 234.283,Z 327.855,A -85,B 0,C 180,E1 19057.698,E2 19057.698} C_VEL
LIN {X 0,Y 231.957,Z 324.652,A -85,B 0,C 180,E1 19064.941,E2 19064.941} C_VEL
LIN {X 0,Y 234.321,Z 327.264,A -85,B 0,C 180,E1 19073.145,E2 19073.145} C_VEL
LIN {X 0,Y 236.235,Z 329.439,A -85,B 0,C 180,E1 19075.866,E2 19075.866} C_VEL
LIN {X 0,Y 239.603,Z 336.177,A -85,B 0,C 180,E1 19080.023,E2 19080.023} C_VEL
LIN {X 0,Y 244.832,Z 349.602,A -85,B 0,C 180,E1 19085.698,E2 19085.698} C_VEL
LIN {X 0,Y 248.595,Z 366.469,A -85,B 0,C 180,E1 19090.957,E2 19090.957} C_VEL
LIN {X 0,Y 249.11,Z 385.929,A -85,B 0,C 180,E1 19096.157,E2 19096.157} C_VEL
LIN {X 0,Y 247.394,Z 393.065,A -85,B 0,C 180,E1 19097.78,E2 19097.78} C_VEL
LIN {X 0,Y 245.209,Z 398.103,A -85,B 0,C 180,E1 19098.814,E2 19098.814} C_VEL
LIN {X 0,Y 236.632,Z 410.241,A -85,B 0,C 180,E1 19101.055,E2 19101.055} C_VEL
LIN {X 0,Y 228.774,Z 419.649,A -85,B 0,C 180,E1 19103.306,E2 19103.306} C_VEL
LIN {X 0,Y 227.998,Z 420.807,A -85,B 0,C 180,E1 19103.727,E2 19103.727} C_VEL
LIN {X 0,Y 219.552,Z 433.719,A -85,B 0,C 180,E1 19110.101,E2 19110.101} C_VEL
LIN {X 0,Y 214.32,Z 440.287,A -85,B 0,C 180,E1 19115.812,E2 19115.812} C_VEL
LIN {X 0,Y 209.774,Z 443.806,A -85,B 0,C 180,E1 19124.002,E2 19124.002} C_VEL
LIN {X 0,Y 208.432,Z 441.862,A -85,B 0,C 180,E1 19131.191,E2 19131.191} C_VEL
LIN {X 0,Y 209.627,Z 434.822,A -85,B 0,C 180,E1 19138.66,E2 19138.66} C_VEL
LIN {X 0,Y 213.037,Z 422.253,A -85,B 0,C 180,E1 19145.854,E2 19145.854} C_VEL
LIN {X 0,Y 218.353,Z 403.391,A -85,B 0,C 180,E1 19152.466,E2 19152.466} C_VEL
LIN {X 0,Y 218.374,Z 401.571,A -85,B 0,C 180,E1 19153.213,E2 19153.213} C_VEL
LIN {X 0,Y 213.968,Z 419.762,A -85,B 0,C 180,E1 19158.818,E2 19158.818} C_VEL
LIN {X 0,Y 210.657,Z 431.992,A -85,B 0,C 180,E1 19164.864,E2 19164.864} C_VEL
LIN {X 0,Y 208.722,Z 439.932,A -85,B 0,C 180,E1 19172.073,E2 19172.073} C_VEL
LIN {X 0,Y 208.633,Z 442.292,A -85,B 0,C 180,E1 19178.319,E2 19178.319} C_VEL
LIN {X 0,Y 210.763,Z 440.336,A -85,B 0,C 180,E1 19185.117,E2 19185.117} C_VEL
LIN {X 0,Y 214.578,Z 433.581,A -85,B 0,C 180,E1 19191.668,E2 19191.668} C_VEL
LIN {X 0,Y 220.511,Z 420.641,A -85,B 0,C 180,E1 19198.158,E2 19198.158} C_VEL
LIN {X 0,Y 226.754,Z 403.779,A -85,B 0,C 180,E1 19203.231,E2 19203.231} C_VEL
LIN {X 0,Y 233.176,Z 381.255,A -85,B 0,C 180,E1 19207.378,E2 19207.378} C_VEL
LIN {X 0,Y 232.166,Z 364.997,A -85,B 0,C 180,E1 19210.17,E2 19210.17} C_VEL
LIN {X 0,Y 225.851,Z 343.324,A -85,B 0,C 180,E1 19213.734,E2 19213.734} C_VEL
LIN {X 0,Y 211.667,Z 315.327,A -85,B 0,C 180,E1 19218.707,E2 19218.707} C_VEL
LIN {X 0,Y 201.783,Z 299.425,A -85,B 0,C 180,E1 19222.594,E2 19222.594} C_VEL
LIN {X 0,Y 201.638,Z 297.81,A -85,B 0,C 180,E1 19222.876,E2 19222.876} C_VEL
LIN {X 0,Y 202.204,Z 297.81,A -85,B 0,C 180,E1 19233.579,E2 19233.579} C_VEL
LIN {X 0,Y 202.886,Z 297.81,A -85,B 0,C 180,E1 19242.664,E2 19242.664} C_VEL
LIN {X 0,Y 203.791,Z 297.81,A -85,B 0,C 180,E1 19251.457,E2 19251.457} C_VEL
LIN {X 0,Y 204.856,Z 297.81,A -85,B 0,C 180,E1 19259.974,E2 19259.974} C_VEL
LIN {X 0,Y 203.875,Z 297.81,A -85,B 0,C 180,E1 19268.486,E2 19268.486} C_VEL
LIN {X 0,Y 202.984,Z 297.81,A -85,B 0,C 180,E1 19277.272,E2 19277.272} C_VEL
LIN {X 0,Y 202.205,Z 297.81,A -85,B 0,C 180,E1 19286.571,E2 19286.571} C_VEL
LIN {X 0,Y 201.837,Z 297.81,A -85,B 0,C 180,E1 19296.702,E2 19296.702} C_VEL
LIN {X 0,Y 223.223,Z 344.297,A -85,B 0,C 180,E1 19302.995,E2 19302.995} C_VEL
LIN {X 0,Y 232.63,Z 374.459,A -85,B 0,C 180,E1 19306.827,E2 19306.827} C_VEL
LIN {X 0,Y 233.759,Z 383.135,A -85,B 0,C 180,E1 19307.918,E2 19307.918} C_VEL
LIN {X 0,Y 226.763,Z 413.002,A -85,B 0,C 180,E1 19311.4,E2 19311.4} C_VEL
LIN {X 0,Y 218.801,Z 440.509,A -85,B 0,C 180,E1 19316.513,E2 19316.513} C_VEL
LIN {X 0,Y 210.544,Z 470.246,A -85,B 0,C 180,E1 19325.097,E2 19325.097} C_VEL
LIN {X 0,Y 207.405,Z 485.689,A -85,B 0,C 180,E1 19331.86,E2 19331.86} C_VEL
LIN {X 0,Y 206.646,Z 495.672,A -85,B 0,C 180,E1 19339.418,E2 19339.418} C_VEL
LIN {X 0,Y 207.546,Z 499.338,A -85,B 0,C 180,E1 19345.829,E2 19345.829} C_VEL
LIN {X 0,Y 208.107,Z 500.288,A -85,B 0,C 180,E1 19349.999,E2 19349.999} C_VEL
LIN {X 0,Y 207.314,Z 500.332,A -85,B 0,C 180,E1 19354.173,E2 19354.173} C_VEL
LIN {X 0,Y 206.356,Z 496.459,A -85,B 0,C 180,E1 19362.671,E2 19362.671} C_VEL
LIN {X 0,Y 208.998,Z 486.156,A -85,B 0,C 180,E1 19372.274,E2 19372.274} C_VEL
LIN {X 0,Y 215.891,Z 471.139,A -85,B 0,C 180,E1 19380.446,E2 19380.446} C_VEL
LIN {X 0,Y 226.359,Z 450.732,A -85,B 0,C 180,E1 19387.466,E2 19387.466} C_VEL
LIN {X 0,Y 238.284,Z 425.732,A -85,B 0,C 180,E1 19392.902,E2 19392.902} C_VEL
LIN {X 0,Y 249.134,Z 398.55,A -85,B 0,C 180,E1 19396.62,E2 19396.62} C_VEL
LIN {X 0,Y 251.955,Z 389.688,A -85,B 0,C 180,E1 19397.534,E2 19397.534} C_VEL
LIN {X 0,Y 247.687,Z 368.594,A -85,B 0,C 180,E1 19402.492,E2 19402.492} C_VEL
LIN {X 0,Y 240.834,Z 351.547,A -85,B 0,C 180,E1 19408.242,E2 19408.242} C_VEL
LIN {X 0,Y 235.379,Z 340.965,A -85,B 0,C 180,E1 19413.757,E2 19413.757} C_VEL
LIN {X 0,Y 232.387,Z 335.382,A -85,B 0,C 180,E1 19418.194,E2 19418.194} C_VEL
LIN {X 0,Y 230.413,Z 332.445,A -85,B 0,C 180,E1 19424.837,E2 19424.837} C_VEL
LIN {X 0,Y 232.129,Z 334.663,A -85,B 0,C 180,E1 19432.553,E2 19432.553} C_VEL
LIN {X 0,Y 233.939,Z 337.02,A -85,B 0,C 180,E1 19435.564,E2 19435.564} C_VEL
LIN {X 0,Y 237.858,Z 346.172,A -85,B 0,C 180,E1 19441.127,E2 19441.127} C_VEL
LIN {X 0,Y 242.28,Z 363.047,A -85,B 0,C 180,E1 19447.628,E2 19447.628} C_VEL
LIN {X 0,Y 243.61,Z 381.113,A -85,B 0,C 180,E1 19452.999,E2 19452.999} C_VEL
LIN {X 0,Y 242.127,Z 393.518,A -85,B 0,C 180,E1 19456.359,E2 19456.359} C_VEL
LIN {X 0,Y 231.667,Z 414.457,A -85,B 0,C 180,E1 19461.525,E2 19461.525} C_VEL
LIN {X 0,Y 227.998,Z 420.807,A -85,B 0,C 180,E1 19463.727,E2 19463.727} C_VEL
LIN {X 0,Y 219.295,Z 429.804,A -85,B 0,C 180,E1 19466.904,E2 19466.904} C_VEL
LIN {X 0,Y 211.723,Z 436.195,A -85,B 0,C 180,E1 19470.003,E2 19470.003} C_VEL
LIN {X 0,Y 211.084,Z 436.922,A -85,B 0,C 180,E1 19470.531,E2 19470.531} C_VEL
LIN {X 0,Y 206.037,Z 442.499,A -85,B 0,C 180,E1 19476.331,E2 19476.331} C_VEL
LIN {X 0,Y 202.703,Z 444.842,A -85,B 0,C 180,E1 19482.104,E2 19482.104} C_VEL
LIN {X 0,Y 200.803,Z 444.04,A -85,B 0,C 180,E1 19488.762,E2 19488.762} C_VEL
LIN {X 0,Y 201.292,Z 437.913,A -85,B 0,C 180,E1 19497.069,E2 19497.069} C_VEL
LIN {X 0,Y 204.401,Z 426.48,A -85,B 0,C 180,E1 19504.678,E2 19504.678} C_VEL
LIN {X 0,Y 209.375,Z 409.561,A -85,B 0,C 180,E1 19511.514,E2 19511.514} C_VEL
LIN {X 0,Y 210.429,Z 405.256,A -85,B 0,C 180,E1 19513.161,E2 19513.161} C_VEL
LIN {X 0,Y 205.978,Z 422.405,A -85,B 0,C 180,E1 19518.914,E2 19518.914} C_VEL
LIN {X 0,Y 202.462,Z 434.742,A -85,B 0,C 180,E1 19525.727,E2 19525.727} C_VEL
LIN {X 0,Y 200.871,Z 441.108,A -85,B 0,C 180,E1 19532.154,E2 19532.154} C_VEL
LIN {X 0,Y 200.851,Z 443.386,A -85,B 0,C 180,E1 19538.643,E2 19538.643} C_VEL
LIN {X 0,Y 202.516,Z 442.13,A -85,B 0,C 180,E1 19544.267,E2 19544.267} C_VEL
LIN {X 0,Y 206.527,Z 435.907,A -85,B 0,C 180,E1 19551.429,E2 19551.429} C_VEL
LIN {X 0,Y 212.498,Z 423.831,A -85,B 0,C 180,E1 19558.186,E2 19558.186} C_VEL
LIN {X 0,Y 219.298,Z 406.901,A -85,B 0,C 180,E1 19563.723,E2 19563.723} C_VEL
LIN {X 0,Y 225.782,Z 386.151,A -85,B 0,C 180,E1 19567.897,E2 19567.897} C_VEL
LIN {X 0,Y 226.775,Z 375.518,A -85,B 0,C 180,E1 19569.717,E2 19569.717} C_VEL
LIN {X 0,Y 222.652,Z 354.01,A -85,B 0,C 180,E1 19573.564,E2 19573.564} C_VEL
LIN {X 0,Y 212.459,Z 330.343,A -85,B 0,C 180,E1 19577.768,E2 19577.768} C_VEL
LIN {X 0,Y 199.499,Z 308.667,A -85,B 0,C 180,E1 19582.869,E2 19582.869} C_VEL
LIN {X 0,Y 193.909,Z 299.162,A -85,B 0,C 180,E1 19585.49,E2 19585.49} C_VEL
LIN {X 0,Y 193.764,Z 297.81,A -85,B 0,C 180,E1 19585.757,E2 19585.757} C_VEL
LIN {X 0,Y 194.027,Z 297.81,A -85,B 0,C 180,E1 19592.151,E2 19592.151} C_VEL
LIN {X 0,Y 194.832,Z 297.81,A -85,B 0,C 180,E1 19601.923,E2 19601.923} C_VEL
LIN {X 0,Y 195.827,Z 297.81,A -85,B 0,C 180,E1 19611.106,E2 19611.106} C_VEL
LIN {X 0,Y 196.937,Z 297.81,A -85,B 0,C 180,E1 19619.973,E2 19619.973} C_VEL
LIN {X 0,Y 195.902,Z 297.81,A -85,B 0,C 180,E1 19628.834,E2 19628.834} C_VEL
LIN {X 0,Y 194.921,Z 297.81,A -85,B 0,C 180,E1 19638.01,E2 19638.01} C_VEL
LIN {X 0,Y 194.082,Z 297.81,A -85,B 0,C 180,E1 19647.777,E2 19647.777} C_VEL
LIN {X 0,Y 193.928,Z 298.196,A -85,B 0,C 180,E1 19654.926,E2 19654.926} C_VEL
LIN {X 0,Y 215.274,Z 343.305,A -85,B 0,C 180,E1 19661.553,E2 19661.553} C_VEL
LIN {X 0,Y 225.056,Z 374.374,A -85,B 0,C 180,E1 19665.742,E2 19665.742} C_VEL
LIN {X 0,Y 226.663,Z 383.762,A -85,B 0,C 180,E1 19667.048,E2 19667.048} C_VEL
LIN {X 0,Y 219.233,Z 414.108,A -85,B 0,C 180,E1 19670.772,E2 19670.772} C_VEL
LIN {X 0,Y 211.095,Z 440.996,A -85,B 0,C 180,E1 19676.049,E2 19676.049} C_VEL
LIN {X 0,Y 203.209,Z 469.421,A -85,B 0,C 180,E1 19684.133,E2 19684.133} C_VEL
LIN {X 0,Y 199.733,Z 484.744,A -85,B 0,C 180,E1 19691.137,E2 19691.137} C_VEL
LIN {X 0,Y 198.746,Z 494.531,A -85,B 0,C 180,E1 19698.859,E2 19698.859} C_VEL
LIN {X 0,Y 199.655,Z 498.257,A -85,B 0,C 180,E1 19705.664,E2 19705.664} C_VEL
LIN {X 0,Y 200.268,Z 499.096,A -85,B 0,C 180,E1 19709.999,E2 19709.999} C_VEL
LIN {X 0,Y 199.425,Z 499.212,A -85,B 0,C 180,E1 19714.338,E2 19714.338} C_VEL
LIN {X 0,Y 198.516,Z 495.452,A -85,B 0,C 180,E1 19723.181,E2 19723.181} C_VEL
LIN {X 0,Y 201.514,Z 485.331,A -85,B 0,C 180,E1 19733.148,E2 19733.148} C_VEL
LIN {X 0,Y 209.546,Z 469.407,A -85,B 0,C 180,E1 19742.078,E2 19742.078} C_VEL
LIN {X 0,Y 220.888,Z 448.77,A -85,B 0,C 180,E1 19749.19,E2 19749.19} C_VEL
LIN {X 0,Y 233.059,Z 424.645,A -85,B 0,C 180,E1 19754.434,E2 19754.434} C_VEL
LIN {X 0,Y 244.914,Z 396.07,A -85,B 0,C 180,E1 19758.284,E2 19758.284} C_VEL
LIN {X 0,Y 246.085,Z 390.946,A -85,B 0,C 180,E1 19758.993,E2 19758.993} C_VEL
LIN {X 0,Y 242.321,Z 371.361,A -85,B 0,C 180,E1 19764.05,E2 19764.05} C_VEL
LIN {X 0,Y 235.8,Z 354.081,A -85,B 0,C 180,E1 19770.687,E2 19770.687} C_VEL
LIN {X 0,Y 231.957,Z 346.868,A -85,B 0,C 180,E1 19775.363,E2 19775.363} C_VEL
LIN {X 0,Y 230.239,Z 342.881,A -85,B 0,C 180,E1 19778.588,E2 19778.588} C_VEL
LIN {X 0,Y 228.517,Z 340.108,A -85,B 0,C 180,E1 19786.661,E2 19786.661} C_VEL
LIN {X 0,Y 231.167,Z 343.65,A -85,B 0,C 180,E1 19794.744,E2 19794.744} C_VEL
LIN {X 0,Y 234.501,Z 353.732,A -85,B 0,C 180,E1 19800.945,E2 19800.945} C_VEL
LIN {X 0,Y 237.492,Z 368.442,A -85,B 0,C 180,E1 19806.865,E2 19806.865} C_VEL
LIN {X 0,Y 237.799,Z 385.982,A -85,B 0,C 180,E1 19812.39,E2 19812.39} C_VEL
LIN {X 0,Y 235.959,Z 396.38,A -85,B 0,C 180,E1 19815.32,E2 19815.32} C_VEL
LIN {X 0,Y 225.385,Z 416.088,A -85,B 0,C 180,E1 19820.396,E2 19820.396} C_VEL
LIN {X 0,Y 215.478,Z 431.202,A -85,B 0,C 180,E1 19826.771,E2 19826.771} C_VEL
LIN {X 0,Y 211.084,Z 436.922,A -85,B 0,C 180,E1 19830.531,E2 19830.531} C_VEL
LIN {X 0,Y 203.355,Z 442.161,A -85,B 0,C 180,E1 19834.638,E2 19834.638} C_VEL
LIN {X 0,Y 196.766,Z 445.197,A -85,B 0,C 180,E1 19838.532,E2 19838.532} C_VEL
LIN {X 0,Y 196.315,Z 445.415,A -85,B 0,C 180,E1 19839.153,E2 19839.153} C_VEL
LIN {X 0,Y 193.643,Z 445.988,A -85,B 0,C 180,E1 19845.467,E2 19845.467} C_VEL
LIN {X 0,Y 192.931,Z 441.842,A -85,B 0,C 180,E1 19854.064,E2 19854.064} C_VEL
LIN {X 0,Y 195.281,Z 432.051,A -85,B 0,C 180,E1 19862.379,E2 19862.379} C_VEL
LIN {X 0,Y 199.748,Z 417.35,A -85,B 0,C 180,E1 19869.662,E2 19869.662} C_VEL
LIN {X 0,Y 202.598,Z 408.274,A -85,B 0,C 180,E1 19872.947,E2 19872.947} C_VEL
LIN {X 0,Y 197.968,Z 424.922,A -85,B 0,C 180,E1 19879.016,E2 19879.016} C_VEL
LIN {X 0,Y 194.678,Z 435.996,A -85,B 0,C 180,E1 19885.556,E2 19885.556} C_VEL
LIN {X 0,Y 193.034,Z 442.278,A -85,B 0,C 180,E1 19892.241,E2 19892.241} C_VEL
LIN {X 0,Y 193.076,Z 444.48,A -85,B 0,C 180,E1 19898.994,E2 19898.994} C_VEL
LIN {X 0,Y 194.883,Z 443.145,A -85,B 0,C 180,E1 19904.839,E2 19904.839} C_VEL
LIN {X 0,Y 199.189,Z 436.834,A -85,B 0,C 180,E1 19912.26,E2 19912.26} C_VEL
LIN {X 0,Y 205.438,Z 424.88,A -85,B 0,C 180,E1 19919.118,E2 19919.118} C_VEL
LIN {X 0,Y 212.749,Z 407.533,A -85,B 0,C 180,E1 19924.908,E2 19924.908} C_VEL
LIN {X 0,Y 219.546,Z 386.63,A -85,B 0,C 180,E1 19929.149,E2 19929.149} C_VEL
LIN {X 0,Y 220.219,Z 376.298,A -85,B 0,C 180,E1 19931.045,E2 19931.045} C_VEL
LIN {X 0,Y 216.266,Z 355.916,A -85,B 0,C 180,E1 19934.925,E2 19934.925} C_VEL
LIN {X 0,Y 206.742,Z 333.331,A -85,B 0,C 180,E1 19939.245,E2 19939.245} C_VEL
LIN {X 0,Y 192.87,Z 310.034,A -85,B 0,C 180,E1 19945.237,E2 19945.237} C_VEL
LIN {X 0,Y 188.022,Z 303.163,A -85,B 0,C 180,E1 19947.685,E2 19947.685} C_VEL
LIN {X 0,Y 185.982,Z 297.81,A -85,B 0,C 180,E1 19949.139,E2 19949.139} C_VEL
LIN {X 0,Y 186.342,Z 297.81,A -85,B 0,C 180,E1 19956.083,E2 19956.083} C_VEL
LIN {X 0,Y 187.285,Z 297.81,A -85,B 0,C 180,E1 19965.982,E2 19965.982} C_VEL
LIN {X 0,Y 188.435,Z 297.81,A -85,B 0,C 180,E1 19975.378,E2 19975.378} C_VEL
LIN {X 0,Y 189.023,Z 297.81,A -85,B 0,C 180,E1 19979.971,E2 19979.971} C_VEL
LIN {X 0,Y 187.9,Z 297.81,A -85,B 0,C 180,E1 19989.214,E2 19989.214} C_VEL
LIN {X 0,Y 186.894,Z 297.81,A -85,B 0,C 180,E1 19998.812,E2 19998.812} C_VEL
LIN {X 0,Y 186.071,Z 297.81,A -85,B 0,C 180,E1 20009.084,E2 20009.084} C_VEL
LIN {X 0,Y 186,Z 298.335,A -85,B 0,C 180,E1 20012.896,E2 20012.896} C_VEL
LIN {X 0,Y 206.739,Z 341.148,A -85,B 0,C 180,E1 20019.83,E2 20019.83} C_VEL
LIN {X 0,Y 216.202,Z 369.393,A -85,B 0,C 180,E1 20023.882,E2 20023.882} C_VEL
LIN {X 0,Y 219.483,Z 384.884,A -85,B 0,C 180,E1 20026.2,E2 20026.2} C_VEL
LIN {X 0,Y 211.711,Z 415.051,A -85,B 0,C 180,E1 20030.096,E2 20030.096} C_VEL
LIN {X 0,Y 203.394,Z 441.457,A -85,B 0,C 180,E1 20035.547,E2 20035.547} C_VEL
LIN {X 0,Y 197.451,Z 463.545,A -85,B 0,C 180,E1 20041.328,E2 20041.328} C_VEL
LIN {X 0,Y 192.927,Z 479.655,A -85,B 0,C 180,E1 20047.977,E2 20047.977} C_VEL
LIN {X 0,Y 190.981,Z 490.297,A -85,B 0,C 180,E1 20055.119,E2 20055.119} C_VEL
LIN {X 0,Y 191.064,Z 495.294,A -85,B 0,C 180,E1 20060.91,E2 20060.91} C_VEL
LIN {X 0,Y 191.733,Z 497.168,A -85,B 0,C 180,E1 20065.485,E2 20065.485} C_VEL
LIN {X 0,Y 192.443,Z 497.907,A -85,B 0,C 180,E1 20069.999,E2 20069.999} C_VEL
LIN {X 0,Y 191.521,Z 498.057,A -85,B 0,C 180,E1 20074.518,E2 20074.518} C_VEL
LIN {X 0,Y 190.667,Z 494.456,A -85,B 0,C 180,E1 20083.733,E2 20083.733} C_VEL
LIN {X 0,Y 194.073,Z 484.526,A -85,B 0,C 180,E1 20094.091,E2 20094.091} C_VEL
LIN {X 0,Y 202.762,Z 468.837,A -85,B 0,C 180,E1 20103.288,E2 20103.288} C_VEL
LIN {X 0,Y 214.735,Z 448.529,A -85,B 0,C 180,E1 20110.542,E2 20110.542} C_VEL
LIN {X 0,Y 228.039,Z 423.634,A -85,B 0,C 180,E1 20116.027,E2 20116.027} C_VEL
LIN {X 0,Y 239.753,Z 396.858,A -85,B 0,C 180,E1 20119.684,E2 20119.684} C_VEL
LIN {X 0,Y 240.021,Z 390.232,A -85,B 0,C 180,E1 20121.074,E2 20121.074} C_VEL
LIN {X 0,Y 236.866,Z 373.803,A -85,B 0,C 180,E1 20125.911,E2 20125.911} C_VEL
LIN {X 0,Y 231.931,Z 359.866,A -85,B 0,C 180,E1 20131.881,E2 20131.881} C_VEL
LIN {X 0,Y 227.96,Z 350.421,A -85,B 0,C 180,E1 20138.672,E2 20138.672} C_VEL
LIN {X 0,Y 226.258,Z 347.683,A -85,B 0,C 180,E1 20146.525,E2 20146.525} C_VEL
LIN {X 0,Y 228.398,Z 351.384,A -85,B 0,C 180,E1 20154.681,E2 20154.681} C_VEL
LIN {X 0,Y 230.775,Z 360.721,A -85,B 0,C 180,E1 20160.582,E2 20160.582} C_VEL
LIN {X 0,Y 232.682,Z 375.03,A -85,B 0,C 180,E1 20166.54,E2 20166.54} C_VEL
LIN {X 0,Y 231.94,Z 390.91,A -85,B 0,C 180,E1 20171.79,E2 20171.79} C_VEL
LIN {X 0,Y 229.78,Z 399.416,A -85,B 0,C 180,E1 20174.28,E2 20174.28} C_VEL
LIN {X 0,Y 218.556,Z 418.904,A -85,B 0,C 180,E1 20179.585,E2 20179.585} C_VEL
LIN {X 0,Y 208.731,Z 432.694,A -85,B 0,C 180,E1 20185.736,E2 20185.736} C_VEL
LIN {X 0,Y 200.996,Z 441.584,A -85,B 0,C 180,E1 20192.718,E2 20192.718} C_VEL
LIN {X 0,Y 196.315,Z 445.415,A -85,B 0,C 180,E1 20199.153,E2 20199.153} C_VEL
LIN {X 0,Y 192.05,Z 446.5,A -85,B 0,C 180,E1 20202.797,E2 20202.797} C_VEL
LIN {X 0,Y 185.271,Z 446.139,A -85,B 0,C 180,E1 20208.44,E2 20208.44} C_VEL
LIN {X 0,Y 185.099,Z 445.887,A -85,B 0,C 180,E1 20209.113,E2 20209.113} C_VEL
LIN {X 0,Y 185.925,Z 438.803,A -85,B 0,C 180,E1 20218.279,E2 20218.279} C_VEL
LIN {X 0,Y 189.602,Z 426.339,A -85,B 0,C 180,E1 20226.552,E2 20226.552} C_VEL
LIN {X 0,Y 194.359,Z 411.593,A -85,B 0,C 180,E1 20232.784,E2 20232.784} C_VEL
LIN {X 0,Y 189.954,Z 427.426,A -85,B 0,C 180,E1 20239.126,E2 20239.126} C_VEL
LIN {X 0,Y 186.467,Z 438.563,A -85,B 0,C 180,E1 20246.522,E2 20246.522} C_VEL
LIN {X 0,Y 185.007,Z 444.567,A -85,B 0,C 180,E1 20254.68,E2 20254.68} C_VEL
LIN {X 0,Y 185.309,Z 445.569,A -85,B 0,C 180,E1 20259.374,E2 20259.374} C_VEL
LIN {X 0,Y 187.705,Z 443.72,A -85,B 0,C 180,E1 20266.343,E2 20266.343} C_VEL
LIN {X 0,Y 192.671,Z 436.397,A -85,B 0,C 180,E1 20274.199,E2 20274.199} C_VEL
LIN {X 0,Y 199.82,Z 423.168,A -85,B 0,C 180,E1 20281.279,E2 20281.279} C_VEL
LIN {X 0,Y 207.033,Z 406.256,A -85,B 0,C 180,E1 20286.656,E2 20286.656} C_VEL
LIN {X 0,Y 214.037,Z 384.779,A -85,B 0,C 180,E1 20290.852,E2 20290.852} C_VEL
LIN {X 0,Y 211.662,Z 363.771,A -85,B 0,C 180,E1 20295.157,E2 20295.157} C_VEL
LIN {X 0,Y 203.668,Z 341.421,A -85,B 0,C 180,E1 20299.724,E2 20299.724} C_VEL
LIN {X 0,Y 189.9,Z 316.883,A -85,B 0,C 180,E1 20306.004,E2 20306.004} C_VEL
LIN {X 0,Y 181.195,Z 304.073,A -85,B 0,C 180,E1 20310.87,E2 20310.87} C_VEL
LIN {X 0,Y 178.299,Z 299.207,A -85,B 0,C 180,E1 20312.814,E2 20312.814} C_VEL
LIN {X 0,Y 178.208,Z 297.81,A -85,B 0,C 180,E1 20313.38,E2 20313.38} C_VEL
LIN {X 0,Y 178.715,Z 297.81,A -85,B 0,C 180,E1 20320.228,E2 20320.228} C_VEL
LIN {X 0,Y 179.805,Z 297.81,A -85,B 0,C 180,E1 20330.307,E2 20330.307} C_VEL
LIN {X 0,Y 181.084,Z 297.81,A -85,B 0,C 180,E1 20340.079,E2 20340.079} C_VEL
LIN {X 0,Y 179.886,Z 297.81,A -85,B 0,C 180,E1 20349.628,E2 20349.628} C_VEL
LIN {X 0,Y 178.784,Z 297.81,A -85,B 0,C 180,E1 20359.7,E2 20359.7} C_VEL
LIN {X 0,Y 178.083,Z 298.595,A -85,B 0,C 180,E1 20370.69,E2 20370.69} C_VEL
LIN {X 0,Y 197.443,Z 337.14,A -85,B 0,C 180,E1 20377.659,E2 20377.659} C_VEL
LIN {X 0,Y 207.882,Z 366.259,A -85,B 0,C 180,E1 20382.147,E2 20382.147} C_VEL
LIN {X 0,Y 212.08,Z 387.161,A -85,B 0,C 180,E1 20385.424,E2 20385.424} C_VEL
LIN {X 0,Y 204.2,Z 415.888,A -85,B 0,C 180,E1 20389.364,E2 20389.364} C_VEL
LIN {X 0,Y 193.326,Z 453.136,A -85,B 0,C 180,E1 20397.212,E2 20397.212} C_VEL
LIN {X 0,Y 187.422,Z 471.971,A -85,B 0,C 180,E1 20403.714,E2 20403.714} C_VEL
LIN {X 0,Y 183.94,Z 484.828,A -85,B 0,C 180,E1 20410.842,E2 20410.842} C_VEL
LIN {X 0,Y 182.95,Z 492.621,A -85,B 0,C 180,E1 20418.099,E2 20418.099} C_VEL
LIN {X 0,Y 183.835,Z 496.083,A -85,B 0,C 180,E1 20425.29,E2 20425.29} C_VEL
LIN {X 0,Y 184.621,Z 496.705,A -85,B 0,C 180,E1 20429.999,E2 20429.999} C_VEL
LIN {X 0,Y 182.973,Z 495.793,A -85,B 0,C 180,E1 20439.493,E2 20439.493} C_VEL
LIN {X 0,Y 184.175,Z 489.003,A -85,B 0,C 180,E1 20450.188,E2 20450.188} C_VEL
LIN {X 0,Y 190.389,Z 477.304,A -85,B 0,C 180,E1 20459.709,E2 20459.709} C_VEL
LIN {X 0,Y 201.262,Z 460.283,A -85,B 0,C 180,E1 20468.007,E2 20468.007} C_VEL
LIN {X 0,Y 214.764,Z 438.115,A -85,B 0,C 180,E1 20474.637,E2 20474.637} C_VEL
LIN {X 0,Y 228.576,Z 411.828,A -85,B 0,C 180,E1 20479.392,E2 20479.392} C_VEL
LIN {X 0,Y 234.78,Z 397.615,A -85,B 0,C 180,E1 20481.161,E2 20481.161} C_VEL
LIN {X 0,Y 232.75,Z 380.955,A -85,B 0,C 180,E1 20486.127,E2 20486.127} C_VEL
LIN {X 0,Y 228.457,Z 366.534,A -85,B 0,C 180,E1 20492.486,E2 20492.486} C_VEL
LIN {X 0,Y 225.218,Z 357.715,A -85,B 0,C 180,E1 20499.035,E2 20499.035} C_VEL
LIN {X 0,Y 223.808,Z 355.351,A -85,B 0,C 180,E1 20504.378,E2 20504.378} C_VEL
LIN {X 0,Y 224.574,Z 357.087,A -85,B 0,C 180,E1 20512.301,E2 20512.301} C_VEL
LIN {X 0,Y 226.04,Z 362.109,A -85,B 0,C 180,E1 20517.116,E2 20517.116} C_VEL
LIN {X 0,Y 227.473,Z 373.835,A -85,B 0,C 180,E1 20523.159,E2 20523.159} C_VEL
LIN {X 0,Y 227.071,Z 389.079,A -85,B 0,C 180,E1 20528.953,E2 20528.953} C_VEL
LIN {X 0,Y 224.243,Z 401.537,A -85,B 0,C 180,E1 20532.965,E2 20532.965} C_VEL
LIN {X 0,Y 212.067,Z 421.161,A -85,B 0,C 180,E1 20538.528,E2 20538.528} C_VEL
LIN {X 0,Y 200.733,Z 435.693,A -85,B 0,C 180,E1 20545.569,E2 20545.569} C_VEL
LIN {X 0,Y 192.505,Z 444.071,A -85,B 0,C 180,E1 20553.313,E2 20553.313} C_VEL
LIN {X 0,Y 187.986,Z 447.029,A -85,B 0,C 180,E1 20559.993,E2 20559.993} C_VEL
LIN {X 0,Y 185.099,Z 445.887,A -85,B 0,C 180,E1 20569.113,E2 20569.113} C_VEL
LIN {X 0,Y 182.517,Z 444.013,A -85,B 0,C 180,E1 20573.093,E2 20573.093} C_VEL
LIN {X 0,Y 178.339,Z 439.104,A -85,B 0,C 180,E1 20579.057,E2 20579.057} C_VEL
LIN {X 0,Y 178.457,Z 438.329,A -85,B 0,C 180,E1 20579.718,E2 20579.718} C_VEL
LIN {X 0,Y 182.433,Z 425.716,A -85,B 0,C 180,E1 20587.854,E2 20587.854} C_VEL
LIN {X 0,Y 186.35,Z 415.139,A -85,B 0,C 180,E1 20592.78,E2 20592.78} C_VEL
LIN {X 0,Y 181.571,Z 430.86,A -85,B 0,C 180,E1 20599.829,E2 20599.829} C_VEL
LIN {X 0,Y 178.29,Z 440.984,A -85,B 0,C 180,E1 20607.576,E2 20607.576} C_VEL
LIN {X 0,Y 177.168,Z 445.701,A -85,B 0,C 180,E1 20614.887,E2 20614.887} C_VEL
LIN {X 0,Y 177.562,Z 446.649,A -85,B 0,C 180,E1 20619.787,E2 20619.787} C_VEL
LIN {X 0,Y 180.179,Z 444.722,A -85,B 0,C 180,E1 20627.047,E2 20627.047} C_VEL
LIN {X 0,Y 185.379,Z 437.46,A -85,B 0,C 180,E1 20635.08,E2 20635.08} C_VEL
LIN {X 0,Y 192.438,Z 425.219,A -85,B 0,C 180,E1 20641.96,E2 20641.96} C_VEL
LIN {X 0,Y 200.123,Z 408.385,A -85,B 0,C 180,E1 20647.621,E2 20647.621} C_VEL
LIN {X 0,Y 207.651,Z 386.338,A -85,B 0,C 180,E1 20652.115,E2 20652.115} C_VEL
LIN {X 0,Y 205.719,Z 366.801,A -85,B 0,C 180,E1 20656.377,E2 20656.377} C_VEL
LIN {X 0,Y 198.486,Z 345.207,A -85,B 0,C 180,E1 20661.119,E2 20661.119} C_VEL
LIN {X 0,Y 186.107,Z 322.734,A -85,B 0,C 180,E1 20667.232,E2 20667.232} C_VEL
LIN {X 0,Y 177.587,Z 310.066,A -85,B 0,C 180,E1 20672.347,E2 20672.347} C_VEL
LIN {X 0,Y 174.006,Z 304.448,A -85,B 0,C 180,E1 20674.949,E2 20674.949} C_VEL
LIN {X 0,Y 170.711,Z 299.664,A -85,B 0,C 180,E1 20677.638,E2 20677.638} C_VEL
LIN {X 0,Y 170.571,Z 297.81,A -85,B 0,C 180,E1 20678.316,E2 20678.316} C_VEL
LIN {X 0,Y 171.365,Z 297.81,A -85,B 0,C 180,E1 20685.617,E2 20685.617} C_VEL
LIN {X 0,Y 172.494,Z 297.81,A -85,B 0,C 180,E1 20694.95,E2 20694.95} C_VEL
LIN {X 0,Y 173.214,Z 297.81,A -85,B 0,C 180,E1 20699.969,E2 20699.969} C_VEL
LIN {X 0,Y 171.862,Z 297.81,A -85,B 0,C 180,E1 20710.082,E2 20710.082} C_VEL
LIN {X 0,Y 170.722,Z 297.81,A -85,B 0,C 180,E1 20720.672,E2 20720.672} C_VEL
LIN {X 0,Y 170.249,Z 298.483,A -85,B 0,C 180,E1 20726.272,E2 20726.272} C_VEL
LIN {X 0,Y 172.479,Z 303.476,A -85,B 0,C 180,E1 20728.337,E2 20728.337} C_VEL
LIN {X 0,Y 174.297,Z 306.349,A -85,B 0,C 180,E1 20729.772,E2 20729.772} C_VEL
LIN {X 0,Y 189.403,Z 336.234,A -85,B 0,C 180,E1 20735.793,E2 20735.793} C_VEL
LIN {X 0,Y 199.828,Z 364.251,A -85,B 0,C 180,E1 20740.456,E2 20740.456} C_VEL
LIN {X 0,Y 205.254,Z 387.059,A -85,B 0,C 180,E1 20744.343,E2 20744.343} C_VEL
LIN {X 0,Y 196.736,Z 416.728,A -85,B 0,C 180,E1 20748.58,E2 20748.58} C_VEL
LIN {X 0,Y 188.48,Z 446.193,A -85,B 0,C 180,E1 20754.222,E2 20754.222} C_VEL
LIN {X 0,Y 182.202,Z 465.464,A -85,B 0,C 180,E1 20760.202,E2 20760.202} C_VEL
LIN {X 0,Y 177.24,Z 480.242,A -85,B 0,C 180,E1 20767.471,E2 20767.471} C_VEL
LIN {X 0,Y 175.091,Z 490.611,A -85,B 0,C 180,E1 20776.289,E2 20776.289} C_VEL
LIN {X 0,Y 175.938,Z 494.997,A -85,B 0,C 180,E1 20785.078,E2 20785.078} C_VEL
LIN {X 0,Y 176.795,Z 495.459,A -85,B 0,C 180,E1 20789.999,E2 20789.999} C_VEL
LIN {X 0,Y 175.064,Z 494.715,A -85,B 0,C 180,E1 20799.926,E2 20799.926} C_VEL
LIN {X 0,Y 176.671,Z 487.96,A -85,B 0,C 180,E1 20811.283,E2 20811.283} C_VEL
LIN {X 0,Y 183.358,Z 476.674,A -85,B 0,C 180,E1 20820.953,E2 20820.953} C_VEL
LIN {X 0,Y 195.423,Z 459.258,A -85,B 0,C 180,E1 20829.719,E2 20829.719} C_VEL
LIN {X 0,Y 209.841,Z 437.015,A -85,B 0,C 180,E1 20836.426,E2 20836.426} C_VEL
LIN {X 0,Y 224.187,Z 411.119,A -85,B 0,C 180,E1 20841.1,E2 20841.1} C_VEL
LIN {X 0,Y 229.117,Z 399.348,A -85,B 0,C 180,E1 20842.753,E2 20842.753} C_VEL
LIN {X 0,Y 227.747,Z 385.248,A -85,B 0,C 180,E1 20847.355,E2 20847.355} C_VEL
LIN {X 0,Y 224.824,Z 373.356,A -85,B 0,C 180,E1 20852.926,E2 20852.926} C_VEL
LIN {X 0,Y 222.525,Z 366.258,A -85,B 0,C 180,E1 20858.127,E2 20858.127} C_VEL
LIN {X 0,Y 220.954,Z 362.812,A -85,B 0,C 180,E1 20864.171,E2 20864.171} C_VEL
LIN {X 0,Y 220.845,Z 362.74,A -85,B 0,C 180,E1 20868.196,E2 20868.196} C_VEL
LIN {X 0,Y 221.868,Z 365.795,A -85,B 0,C 180,E1 20874.169,E2 20874.169} C_VEL
LIN {X 0,Y 222.765,Z 375.683,A -85,B 0,C 180,E1 20880.603,E2 20880.603} C_VEL
LIN {X 0,Y 222.246,Z 388.75,A -85,B 0,C 180,E1 20886.263,E2 20886.263} C_VEL
LIN {X 0,Y 219.182,Z 403.05,A -85,B 0,C 180,E1 20891.442,E2 20891.442} C_VEL
LIN {X 0,Y 206.432,Z 422.435,A -85,B 0,C 180,E1 20897.029,E2 20897.029} C_VEL
LIN {X 0,Y 195.128,Z 436.122,A -85,B 0,C 180,E1 20903.689,E2 20903.689} C_VEL
LIN {X 0,Y 186.939,Z 444.092,A -85,B 0,C 180,E1 20910.621,E2 20910.621} C_VEL
LIN {X 0,Y 182.989,Z 447.023,A -85,B 0,C 180,E1 20915.295,E2 20915.295} C_VEL
LIN {X 0,Y 178.946,Z 448.448,A -85,B 0,C 180,E1 20922.467,E2 20922.467} C_VEL
LIN {X 0,Y 177.097,Z 445.43,A -85,B 0,C 180,E1 20931.753,E2 20931.753} C_VEL
LIN {X 0,Y 178.457,Z 438.329,A -85,B 0,C 180,E1 20939.718,E2 20939.718} C_VEL
LIN {X 0,Y 178.204,Z 435.152,A -85,B 0,C 180,E1 20942.339,E2 20942.339} C_VEL
LIN {X 0,Y 175.531,Z 424.726,A -85,B 0,C 180,E1 20949.392,E2 20949.392} C_VEL
LIN {X 0,Y 175.85,Z 423.52,A -85,B 0,C 180,E1 20949.983,E2 20949.983} C_VEL
LIN {X 0,Y 177.961,Z 418.188,A -85,B 0,C 180,E1 20952.558,E2 20952.558} C_VEL
LIN {X 0,Y 174.257,Z 431.137,A -85,B 0,C 180,E1 20958.766,E2 20958.766} C_VEL
LIN {X 0,Y 170.457,Z 442.198,A -85,B 0,C 180,E1 20967.465,E2 20967.465} C_VEL
LIN {X 0,Y 169.337,Z 446.835,A -85,B 0,C 180,E1 20975.114,E2 20975.114} C_VEL
LIN {X 0,Y 170.711,Z 447.375,A -85,B 0,C 180,E1 20983.363,E2 20983.363} C_VEL
LIN {X 0,Y 174.788,Z 443.203,A -85,B 0,C 180,E1 20991.527,E2 20991.527} C_VEL
LIN {X 0,Y 181.815,Z 432.81,A -85,B 0,C 180,E1 20999.868,E2 20999.868} C_VEL
LIN {X 0,Y 190.097,Z 417.556,A -85,B 0,C 180,E1 21006.49,E2 21006.49} C_VEL
LIN {X 0,Y 198.494,Z 397.358,A -85,B 0,C 180,E1 21011.699,E2 21011.699} C_VEL
LIN {X 0,Y 201.372,Z 386.697,A -85,B 0,C 180,E1 21013.752,E2 21013.752} C_VEL
LIN {X 0,Y 199.28,Z 367.282,A -85,B 0,C 180,E1 21018.25,E2 21018.25} C_VEL
LIN {X 0,Y 192.24,Z 346.401,A -85,B 0,C 180,E1 21023.222,E2 21023.222} C_VEL
LIN {X 0,Y 179.623,Z 323.8,A -85,B 0,C 180,E1 21030.212,E2 21030.212} C_VEL
LIN {X 0,Y 171.123,Z 311.16,A -85,B 0,C 180,E1 21036.241,E2 21036.241} C_VEL
LIN {X 0,Y 166.845,Z 304.697,A -85,B 0,C 180,E1 21040.139,E2 21040.139} C_VEL
LIN {X 0,Y 163.475,Z 300.015,A -85,B 0,C 180,E1 21043.888,E2 21043.888} C_VEL
LIN {X 0,Y 163.346,Z 297.81,A -85,B 0,C 180,E1 21044.895,E2 21044.895} C_VEL
LIN {X 0,Y 164.512,Z 297.81,A -85,B 0,C 180,E1 21054.704,E2 21054.704} C_VEL
LIN {X 0,Y 165.298,Z 297.81,A -85,B 0,C 180,E1 21059.967,E2 21059.967} C_VEL
LIN {X 0,Y 163.885,Z 297.81,A -85,B 0,C 180,E1 21070.579,E2 21070.579} C_VEL
LIN {X 0,Y 162.86,Z 298.545,A -85,B 0,C 180,E1 21079.591,E2 21079.591} C_VEL
LIN {X 0,Y 165.486,Z 303.928,A -85,B 0,C 180,E1 21082.944,E2 21082.944} C_VEL
LIN {X 0,Y 167.858,Z 306.382,A -85,B 0,C 180,E1 21085.243,E2 21085.243} C_VEL
LIN {X 0,Y 172.125,Z 314.48,A -85,B 0,C 180,E1 21089.103,E2 21089.103} C_VEL
LIN {X 0,Y 177.202,Z 326.437,A -85,B 0,C 180,E1 21092.04,E2 21092.04} C_VEL
LIN {X 0,Y 189.542,Z 355.285,A -85,B 0,C 180,E1 21097.393,E2 21097.393} C_VEL
LIN {X 0,Y 196.993,Z 382.883,A -85,B 0,C 180,E1 21102.361,E2 21102.361} C_VEL
LIN {X 0,Y 197.399,Z 390.766,A -85,B 0,C 180,E1 21103.67,E2 21103.67} C_VEL
LIN {X 0,Y 185.118,Z 435.632,A -85,B 0,C 180,E1 21110.481,E2 21110.481} C_VEL
LIN {X 0,Y 178.218,Z 456.417,A -85,B 0,C 180,E1 21115.877,E2 21115.877} C_VEL
LIN {X 0,Y 171.871,Z 473.312,A -85,B 0,C 180,E1 21122.869,E2 21122.869} C_VEL
LIN {X 0,Y 167.779,Z 486.379,A -85,B 0,C 180,E1 21132.046,E2 21132.046} C_VEL
LIN {X 0,Y 167.303,Z 492.147,A -85,B 0,C 180,E1 21139.606,E2 21139.606} C_VEL
LIN {X 0,Y 168.026,Z 493.91,A -85,B 0,C 180,E1 21144.846,E2 21144.846} C_VEL
LIN {X 0,Y 168.964,Z 494.204,A -85,B 0,C 180,E1 21149.999,E2 21149.999} C_VEL
LIN {X 0,Y 167.172,Z 493.641,A -85,B 0,C 180,E1 21160.399,E2 21160.399} C_VEL
LIN {X 0,Y 169.126,Z 487.1,A -85,B 0,C 180,E1 21172.282,E2 21172.282} C_VEL
LIN {X 0,Y 177.764,Z 474.245,A -85,B 0,C 180,E1 21183.487,E2 21183.487} C_VEL
LIN {X 0,Y 190.995,Z 456.589,A -85,B 0,C 180,E1 21192.186,E2 21192.186} C_VEL
LIN {X 0,Y 206.008,Z 434.71,A -85,B 0,C 180,E1 21198.587,E2 21198.587} C_VEL
LIN {X 0,Y 221.178,Z 408.044,A -85,B 0,C 180,E1 21203.201,E2 21203.201} C_VEL
LIN {X 0,Y 223.602,Z 402.367,A -85,B 0,C 180,E1 21204.077,E2 21204.077} C_VEL
LIN {X 0,Y 222.689,Z 388.819,A -85,B 0,C 180,E1 21208.942,E2 21208.942} C_VEL
LIN {X 0,Y 220.408,Z 377.912,A -85,B 0,C 180,E1 21214.691,E2 21214.691} C_VEL
LIN {X 0,Y 218.701,Z 372.094,A -85,B 0,C 180,E1 21219.844,E2 21219.844} C_VEL
LIN {X 0,Y 217.489,Z 369.935,A -85,B 0,C 180,E1 21226.249,E2 21226.249} C_VEL
LIN {X 0,Y 217.941,Z 371.438,A -85,B 0,C 180,E1 21232.065,E2 21232.065} C_VEL
LIN {X 0,Y 218.312,Z 376.834,A -85,B 0,C 180,E1 21237.053,E2 21237.053} C_VEL
LIN {X 0,Y 217.786,Z 387.903,A -85,B 0,C 180,E1 21243.004,E2 21243.004} C_VEL
LIN {X 0,Y 214.766,Z 402.222,A -85,B 0,C 180,E1 21248.778,E2 21248.778} C_VEL
LIN {X 0,Y 212.071,Z 408.194,A -85,B 0,C 180,E1 21250.702,E2 21250.702} C_VEL
LIN {X 0,Y 198.087,Z 427.284,A -85,B 0,C 180,E1 21256.866,E2 21256.866} C_VEL
LIN {X 0,Y 186.511,Z 439.72,A -85,B 0,C 180,E1 21263.894,E2 21263.894} C_VEL
LIN {X 0,Y 177.728,Z 447.049,A -85,B 0,C 180,E1 21271.894,E2 21271.894} C_VEL
LIN {X 0,Y 173.091,Z 449.394,A -85,B 0,C 180,E1 21278.318,E2 21278.318} C_VEL
LIN {X 0,Y 169.581,Z 448.289,A -85,B 0,C 180,E1 21287.923,E2 21287.923} C_VEL
LIN {X 0,Y 170.052,Z 441.533,A -85,B 0,C 180,E1 21297.832,E2 21297.832} C_VEL
LIN {X 0,Y 173.904,Z 429.168,A -85,B 0,C 180,E1 21307.004,E2 21307.004} C_VEL
LIN {X 0,Y 175.85,Z 423.52,A -85,B 0,C 180,E1 21309.983,E2 21309.983} C_VEL
LIN {X 0,Y 175.326,Z 422.269,A -85,B 0,C 180,E1 21312.16,E2 21312.16} C_VEL
LIN {X 0,Y 171.537,Z 426.221,A -85,B 0,C 180,E1 21315.333,E2 21315.333} C_VEL
LIN {X 0,Y 165.319,Z 435.94,A -85,B 0,C 180,E1 21320.55,E2 21320.55} C_VEL
LIN {X 0,Y 162.056,Z 445.401,A -85,B 0,C 180,E1 21330.002,E2 21330.002} C_VEL
LIN {X 0,Y 161.504,Z 447.969,A -85,B 0,C 180,E1 21335.363,E2 21335.363} C_VEL
LIN {X 0,Y 162.101,Z 448.796,A -85,B 0,C 180,E1 21340.731,E2 21340.731} C_VEL
LIN {X 0,Y 165.181,Z 446.715,A -85,B 0,C 180,E1 21348.649,E2 21348.649} C_VEL
LIN {X 0,Y 171.595,Z 438.728,A -85,B 0,C 180,E1 21357.749,E2 21357.749} C_VEL
LIN {X 0,Y 179.955,Z 425.497,A -85,B 0,C 180,E1 21365.206,E2 21365.206} C_VEL
LIN {X 0,Y 188.973,Z 407.066,A -85,B 0,C 180,E1 21371.209,E2 21371.209} C_VEL
LIN {X 0,Y 195.148,Z 389.43,A -85,B 0,C 180,E1 21374.906,E2 21374.906} C_VEL
LIN {X 0,Y 193.622,Z 370.818,A -85,B 0,C 180,E1 21379.512,E2 21379.512} C_VEL
LIN {X 0,Y 187.064,Z 349.732,A -85,B 0,C 180,E1 21384.94,E2 21384.94} C_VEL
LIN {X 0,Y 175.541,Z 328.85,A -85,B 0,C 180,E1 21391.996,E2 21391.996} C_VEL
LIN {X 0,Y 168.178,Z 317.549,A -85,B 0,C 180,E1 21397.722,E2 21397.722} C_VEL
LIN {X 0,Y 164.548,Z 311.868,A -85,B 0,C 180,E1 21401.323,E2 21401.323} C_VEL
LIN {X 0,Y 161.267,Z 306.134,A -85,B 0,C 180,E1 21405.469,E2 21405.469} C_VEL
LIN {X 0,Y 156.753,Z 300.049,A -85,B 0,C 180,E1 21414.095,E2 21414.095} C_VEL
LIN {X 0,Y 156.689,Z 297.81,A -85,B 0,C 180,E1 21415.823,E2 21415.823} C_VEL
LIN {X 0,Y 157.361,Z 297.81,A -85,B 0,C 180,E1 21419.966,E2 21419.966} C_VEL
LIN {X 0,Y 156.172,Z 298.227,A -85,B 0,C 180,E1 21427.775,E2 21427.775} C_VEL
LIN {X 0,Y 158.57,Z 304.158,A -85,B 0,C 180,E1 21434.864,E2 21434.864} C_VEL
LIN {X 0,Y 160.985,Z 306.181,A -85,B 0,C 180,E1 21438.555,E2 21438.555} C_VEL
LIN {X 0,Y 164.332,Z 311.869,A -85,B 0,C 180,E1 21442.847,E2 21442.847} C_VEL
LIN {X 0,Y 168.748,Z 319.267,A -85,B 0,C 180,E1 21447.238,E2 21447.238} C_VEL
LIN {X 0,Y 174.951,Z 337.155,A -85,B 0,C 180,E1 21452.101,E2 21452.101} C_VEL
LIN {X 0,Y 185.481,Z 365.967,A -85,B 0,C 180,E1 21457.741,E2 21457.741} C_VEL
LIN {X 0,Y 190.622,Z 390.61,A -85,B 0,C 180,E1 21462.478,E2 21462.478} C_VEL
LIN {X 0,Y 181.2,Z 427.76,A -85,B 0,C 180,E1 21467.417,E2 21467.417} C_VEL
LIN {X 0,Y 173.744,Z 450.005,A -85,B 0,C 180,E1 21472.556,E2 21472.556} C_VEL
LIN {X 0,Y 166.067,Z 469.136,A -85,B 0,C 180,E1 21479.863,E2 21479.863} C_VEL
LIN {X 0,Y 161.087,Z 481.928,A -85,B 0,C 180,E1 21487.992,E2 21487.992} C_VEL
LIN {X 0,Y 159.345,Z 489.515,A -85,B 0,C 180,E1 21496.304,E2 21496.304} C_VEL
LIN {X 0,Y 160.117,Z 492.822,A -85,B 0,C 180,E1 21504.591,E2 21504.591} C_VEL
LIN {X 0,Y 161.141,Z 492.93,A -85,B 0,C 180,E1 21509.998,E2 21509.998} C_VEL
LIN {X 0,Y 159.272,Z 492.561,A -85,B 0,C 180,E1 21520.921,E2 21520.921} C_VEL
LIN {X 0,Y 161.641,Z 486.231,A -85,B 0,C 180,E1 21533.374,E2 21533.374} C_VEL
LIN {X 0,Y 171.088,Z 473.7,A -85,B 0,C 180,E1 21544.979,E2 21544.979} C_VEL
LIN {X 0,Y 185.139,Z 456.378,A -85,B 0,C 180,E1 21553.851,E2 21553.851} C_VEL
LIN {X 0,Y 200.847,Z 434.882,A -85,B 0,C 180,E1 21560.285,E2 21560.285} C_VEL
LIN {X 0,Y 216.646,Z 408.799,A -85,B 0,C 180,E1 21564.883,E2 21564.883} C_VEL
LIN {X 0,Y 218.157,Z 404.904,A -85,B 0,C 180,E1 21565.596,E2 21565.596} C_VEL
LIN {X 0,Y 217.772,Z 393.247,A -85,B 0,C 180,E1 21570.22,E2 21570.22} C_VEL
LIN {X 0,Y 216.066,Z 382.907,A -85,B 0,C 180,E1 21576.325,E2 21576.325} C_VEL
LIN {X 0,Y 214.618,Z 378.349,A -85,B 0,C 180,E1 21581.581,E2 21581.581} C_VEL
LIN {X 0,Y 214.013,Z 376.978,A -85,B 0,C 180,E1 21587.813,E2 21587.813} C_VEL
LIN {X 0,Y 214.224,Z 380.111,A -85,B 0,C 180,E1 21594.106,E2 21594.106} C_VEL
LIN {X 0,Y 213.416,Z 388.927,A -85,B 0,C 180,E1 21600.025,E2 21600.025} C_VEL
LIN {X 0,Y 210.469,Z 402.128,A -85,B 0,C 180,E1 21606.13,E2 21606.13} C_VEL
LIN {X 0,Y 207.102,Z 410.081,A -85,B 0,C 180,E1 21609.106,E2 21609.106} C_VEL
LIN {X 0,Y 193.017,Z 428.17,A -85,B 0,C 180,E1 21615.004,E2 21615.004} C_VEL
LIN {X 0,Y 179.869,Z 441.335,A -85,B 0,C 180,E1 21622.659,E2 21622.659} C_VEL
LIN {X 0,Y 172.412,Z 447.193,A -85,B 0,C 180,E1 21628.931,E2 21628.931} C_VEL
LIN {X 0,Y 166.873,Z 450.238,A -85,B 0,C 180,E1 21635.529,E2 21635.529} C_VEL
LIN {X 0,Y 163.256,Z 450.669,A -85,B 0,C 180,E1 21642.318,E2 21642.318} C_VEL
LIN {X 0,Y 161.44,Z 447.441,A -85,B 0,C 180,E1 21651.5,E2 21651.5} C_VEL
LIN {X 0,Y 163.271,Z 438.804,A -85,B 0,C 180,E1 21661.372,E2 21661.372} C_VEL
LIN {X 0,Y 168.328,Z 424.209,A -85,B 0,C 180,E1 21670.731,E2 21670.731} C_VEL
LIN {X 0,Y 169.889,Z 421.493,A -85,B 0,C 180,E1 21672.536,E2 21672.536} C_VEL
LIN {X 0,Y 167.867,Z 429.164,A -85,B 0,C 180,E1 21676.353,E2 21676.353} C_VEL
LIN {X 0,Y 165.319,Z 435.94,A -85,B 0,C 180,E1 21680.55,E2 21680.55} C_VEL
LIN {X 0,Y 161.072,Z 441.288,A -85,B 0,C 180,E1 21684.493,E2 21684.493} C_VEL
LIN {X 0,Y 154.135,Z 447.089,A -85,B 0,C 180,E1 21690.928,E2 21690.928} C_VEL
LIN {X 0,Y 153.937,Z 447.484,A -85,B 0,C 180,E1 21691.727,E2 21691.727} C_VEL
LIN {X 0,Y 154.778,Z 449.801,A -85,B 0,C 180,E1 21702.688,E2 21702.688} C_VEL
LIN {X 0,Y 159.326,Z 446.092,A -85,B 0,C 180,E1 21712.264,E2 21712.264} C_VEL
LIN {X 0,Y 166.093,Z 437.639,A -85,B 0,C 180,E1 21720.514,E2 21720.514} C_VEL
LIN {X 0,Y 175.623,Z 422.62,A -85,B 0,C 180,E1 21728.197,E2 21728.197} C_VEL
LIN {X 0,Y 184.996,Z 403.22,A -85,B 0,C 180,E1 21733.897,E2 21733.897} C_VEL
LIN {X 0,Y 189.062,Z 391.389,A -85,B 0,C 180,E1 21736.331,E2 21736.331} C_VEL
LIN {X 0,Y 187.823,Z 373.167,A -85,B 0,C 180,E1 21741.159,E2 21741.159} C_VEL
LIN {X 0,Y 181.948,Z 353.204,A -85,B 0,C 180,E1 21746.756,E2 21746.756} C_VEL
LIN {X 0,Y 172.03,Z 334.316,A -85,B 0,C 180,E1 21753.59,E2 21753.59} C_VEL
LIN {X 0,Y 165.167,Z 323.431,A -85,B 0,C 180,E1 21759.461,E2 21759.461} C_VEL
LIN {X 0,Y 162.026,Z 318.581,A -85,B 0,C 180,E1 21762.895,E2 21762.895} C_VEL
LIN {X 0,Y 158.618,Z 312.53,A -85,B 0,C 180,E1 21767.821,E2 21767.821} C_VEL
LIN {X 0,Y 155.479,Z 307.37,A -85,B 0,C 180,E1 21775.093,E2 21775.093} C_VEL
LIN {X 0,Y 155.112,Z 305.523,A -85,B 0,C 180,E1 21777.177,E2 21777.177} C_VEL
LIN {X 0,Y 155.01,Z 306.294,A -85,B 0,C 180,E1 21787.13,E2 21787.13} C_VEL
LIN {X 0,Y 157.854,Z 312.283,A -85,B 0,C 180,E1 21795.356,E2 21795.356} C_VEL
LIN {X 0,Y 159.513,Z 314.455,A -85,B 0,C 180,E1 21798.05,E2 21798.05} C_VEL
LIN {X 0,Y 164.119,Z 322.072,A -85,B 0,C 180,E1 21803.864,E2 21803.864} C_VEL
LIN {X 0,Y 166.49,Z 327.291,A -85,B 0,C 180,E1 21806.368,E2 21806.368} C_VEL
LIN {X 0,Y 176.202,Z 359.563,A -85,B 0,C 180,E1 21814.717,E2 21814.717} C_VEL
LIN {X 0,Y 183.25,Z 388.033,A -85,B 0,C 180,E1 21820.584,E2 21820.584} C_VEL
LIN {X 0,Y 183.383,Z 394,A -85,B 0,C 180,E1 21821.413,E2 21821.413} C_VEL
LIN {X 0,Y 177.895,Z 419.146,A -85,B 0,C 180,E1 21824.296,E2 21824.296} C_VEL
LIN {X 0,Y 169.991,Z 442.587,A -85,B 0,C 180,E1 21828.976,E2 21828.976} C_VEL
LIN {X 0,Y 162.098,Z 461.502,A -85,B 0,C 180,E1 21835.235,E2 21835.235} C_VEL
LIN {X 0,Y 155.028,Z 477.436,A -85,B 0,C 180,E1 21844.021,E2 21844.021} C_VEL
LIN {X 0,Y 151.643,Z 487.555,A -85,B 0,C 180,E1 21854.117,E2 21854.117} C_VEL
LIN {X 0,Y 152.193,Z 491.732,A -85,B 0,C 180,E1 21864.308,E2 21864.308} C_VEL
LIN {X 0,Y 153.296,Z 491.653,A -85,B 0,C 180,E1 21869.998,E2 21869.998} C_VEL
LIN {X 0,Y 151.384,Z 491.435,A -85,B 0,C 180,E1 21881.498,E2 21881.498} C_VEL
LIN {X 0,Y 153.538,Z 486.299,A -85,B 0,C 180,E1 21893.147,E2 21893.147} C_VEL
LIN {X 0,Y 163.013,Z 474.774,A -85,B 0,C 180,E1 21905.347,E2 21905.347} C_VEL
LIN {X 0,Y 177.301,Z 458.626,A -85,B 0,C 180,E1 21914.598,E2 21914.598} C_VEL
LIN {X 0,Y 194.23,Z 437.38,A -85,B 0,C 180,E1 21921.526,E2 21921.526} C_VEL
